// TwinCAT 3 PLC project PLC_Light_Control
// ProgramVersion: 3.1.4023.0
// libraries:
//   Tc2_BABasic, * (Beckhoff Automation GmbH)
//   Tc2_BACnetRev12, * (Beckhoff Automation GmbH)
//   Tc2_DALI, * (Beckhoff Automation GmbH)
//   Tc2_EIB, * (Beckhoff Automation GmbH)
//   Tc2_Standard, * (Beckhoff Automation GmbH)
//   Tc2_System, * (Beckhoff Automation GmbH)
//   Tc2_Utilities, * (Beckhoff Automation GmbH)
//   Tc3_Module, * (Beckhoff Automation GmbH)
// project tree:
//   / CommunicationTask.TcTTO, DimmerTask.TcTTO, PlcTask.TcTTO
//   DUTs/ E_KL6821Module.TcDUT, ST_DALI_Lamp.TcDUT
//   GVLs/ GVL_BACnet.TcGVL, GVL_GenSysInfo.TcGVL, GVL_IO.TcGVL, GVL_StreetLamps.TcGVL
//   POUs/BACnetControl/ P_BACnet_ActualLevel.TcPOU, P_BACnet_Error.TcPOU, P_BACnet_Level.TcPOU, P_BACnet_Manual.TcPOU, P_BACnet_Motion.TcPOU, P_BACnet_Scene.TcPOU
//   POUs/DimmersStreetLamps/ P_Dimmers_RB1.TcPOU, P_Dimmers_Broadcast.TcPOU, P_Dimmers_RB2.TcPOU, P_Dimmers_RB3.TcPOU
//   POUs/ FB_PBL.TcPOU, FB_SceneController.TcPOU, F_IsNight.TcPOU, MAIN.TcPOU, P_AddrAssignment.TcPOU, P_AlarmMode.TcPOU, P_AutoMode.TcPOU, P_AutoMode_Old_Broadcast.TcPOU
//   POUs/KL6821Communication/ P_DALI_RB1_Communication.TcPOU, P_DALI_RB2_Communication.TcPOU, P_DALI_RB3_Communication.TcPOU
//   POUs/KNX/ P_KNX_Communication.TcPOU, P_KNX_Data_GatesANDAlarm.TcPOU, P_KNX_Data_MotionSensors.TcPOU, P_MotionSensors.TcPOU
// real-time tasks:
//   TASK PlcTask: cycle T#10ms, priority 20, ADS port 350
//   TASK CommunicationTask: cycle T#2ms, priority 7, ADS port 351
//   TASK DimmerTask: cycle T#10ms, priority 15, ADS port 352
//   TASK Device 1 (BACnet IP)_Task_58: cycle T#40ms, priority 58, ADS port 353
//   TASK Device 1 (BACnet IP)_QueueTask: cycle T#2ms, priority 8, ADS port 354
// I/O:
//   DEVICE Device 1 (BACnet IP), AmsNetId 26.242.21.199.2.1
// variable links:
//   PLC_Light_Control Instance <-> Device 1 (BACnet IP)
//     CommunicationTask Inputs/Tc2_BACnetRev12.BACnet_Globals.fbBACnet_Adapter._AmsNetId <-> Inputs/AmsNetId
//     CommunicationTask Inputs/Tc2_BACnetRev12.BACnet_Globals.fbBACnet_Adapter._DeviceStatus <-> Inputs/Device Status
//   PLC_Light_Control Instance <-> Device 1 (BACnet IP)/Beckhoff_496669 (BACnet Server)
//     CommunicationTask Inputs/GVL_BACnet.Device._ServerStatus <-> Inputs/Server Status
//     CommunicationTask Outputs/GVL_BACnet.Device._ServerControl <-> Outputs/Server Control
//   PLC_Light_Control Instance <-> Device 1 (BACnet IP)/Beckhoff_496669 (BACnet Server)/Beckhoff_496669 (BACnet Device Object)
//     CommunicationTask Inputs/GVL_BACnet.Device._LocalDate <-> Inputs/LocalDate
//     CommunicationTask Inputs/GVL_BACnet.Device._LocalTime <-> Inputs/LocalTime
//     CommunicationTask Inputs/GVL_BACnet.Device._ObjectId <-> Inputs/ObjectIdentifier
//     CommunicationTask Inputs/GVL_BACnet.Device._SystemStatus <-> Inputs/SystemStatus
//   PLC_Light_Control Instance <-> Device 1 (BACnet IP)/Beckhoff_496669 (BACnet Server)/GVL_BACnet (BACnet Structured View Object)/fbBACnet_AV_Gates (BACnet Analog Value Object)
//     CommunicationTask Inputs/GVL_BACnet.fbBACnet_AV_Gates._PresentValue <-> Inputs/PresentValue
//     CommunicationTask Inputs/GVL_BACnet.fbBACnet_AV_Gates._StatusFlags <-> Inputs/StatusFlags
//     CommunicationTask Outputs/GVL_BACnet.fbBACnet_AV_Gates._PresentValue_Priority12 <-> Outputs/PresentValue_Priority12
//   PLC_Light_Control Instance <-> Device 1 (BACnet IP)/Beckhoff_496669 (BACnet Server)/GVL_BACnet (BACnet Structured View Object)/fbBACnet_AV_SL_ActualLevel_1 (BACnet Analog Value Object)
//     PlcTask Inputs/GVL_BACnet.fbBACnet_AV_SL_ActualLevel_1._PresentValue <-> Inputs/PresentValue
//     PlcTask Inputs/GVL_BACnet.fbBACnet_AV_SL_ActualLevel_1._StatusFlags <-> Inputs/StatusFlags
//     PlcTask Outputs/GVL_BACnet.fbBACnet_AV_SL_ActualLevel_1._PresentValue_Priority12 <-> Outputs/PresentValue_Priority12
//   PLC_Light_Control Instance <-> Device 1 (BACnet IP)/Beckhoff_496669 (BACnet Server)/GVL_BACnet (BACnet Structured View Object)/fbBACnet_AV_SL_ActualLevel_10 (BACnet Analog Value Object)
//     PlcTask Inputs/GVL_BACnet.fbBACnet_AV_SL_ActualLevel_10._PresentValue <-> Inputs/PresentValue
//     PlcTask Inputs/GVL_BACnet.fbBACnet_AV_SL_ActualLevel_10._StatusFlags <-> Inputs/StatusFlags
//     PlcTask Outputs/GVL_BACnet.fbBACnet_AV_SL_ActualLevel_10._PresentValue_Priority12 <-> Outputs/PresentValue_Priority12
//   PLC_Light_Control Instance <-> Device 1 (BACnet IP)/Beckhoff_496669 (BACnet Server)/GVL_BACnet (BACnet Structured View Object)/fbBACnet_AV_SL_ActualLevel_2 (BACnet Analog Value Object)
//     PlcTask Inputs/GVL_BACnet.fbBACnet_AV_SL_ActualLevel_2._PresentValue <-> Inputs/PresentValue
//     PlcTask Inputs/GVL_BACnet.fbBACnet_AV_SL_ActualLevel_2._StatusFlags <-> Inputs/StatusFlags
//     PlcTask Outputs/GVL_BACnet.fbBACnet_AV_SL_ActualLevel_2._PresentValue_Priority12 <-> Outputs/PresentValue_Priority12
//   PLC_Light_Control Instance <-> Device 1 (BACnet IP)/Beckhoff_496669 (BACnet Server)/GVL_BACnet (BACnet Structured View Object)/fbBACnet_AV_SL_ActualLevel_3 (BACnet Analog Value Object)
//     PlcTask Inputs/GVL_BACnet.fbBACnet_AV_SL_ActualLevel_3._PresentValue <-> Inputs/PresentValue
//     PlcTask Inputs/GVL_BACnet.fbBACnet_AV_SL_ActualLevel_3._StatusFlags <-> Inputs/StatusFlags
//     PlcTask Outputs/GVL_BACnet.fbBACnet_AV_SL_ActualLevel_3._PresentValue_Priority12 <-> Outputs/PresentValue_Priority12
//   PLC_Light_Control Instance <-> Device 1 (BACnet IP)/Beckhoff_496669 (BACnet Server)/GVL_BACnet (BACnet Structured View Object)/fbBACnet_AV_SL_ActualLevel_4 (BACnet Analog Value Object)
//     PlcTask Inputs/GVL_BACnet.fbBACnet_AV_SL_ActualLevel_4._PresentValue <-> Inputs/PresentValue
//     PlcTask Inputs/GVL_BACnet.fbBACnet_AV_SL_ActualLevel_4._StatusFlags <-> Inputs/StatusFlags
//     PlcTask Outputs/GVL_BACnet.fbBACnet_AV_SL_ActualLevel_4._PresentValue_Priority12 <-> Outputs/PresentValue_Priority12
//   PLC_Light_Control Instance <-> Device 1 (BACnet IP)/Beckhoff_496669 (BACnet Server)/GVL_BACnet (BACnet Structured View Object)/fbBACnet_AV_SL_ActualLevel_5 (BACnet Analog Value Object)
//     PlcTask Inputs/GVL_BACnet.fbBACnet_AV_SL_ActualLevel_5._PresentValue <-> Inputs/PresentValue
//     PlcTask Inputs/GVL_BACnet.fbBACnet_AV_SL_ActualLevel_5._StatusFlags <-> Inputs/StatusFlags
//     PlcTask Outputs/GVL_BACnet.fbBACnet_AV_SL_ActualLevel_5._PresentValue_Priority12 <-> Outputs/PresentValue_Priority12
//   PLC_Light_Control Instance <-> Device 1 (BACnet IP)/Beckhoff_496669 (BACnet Server)/GVL_BACnet (BACnet Structured View Object)/fbBACnet_AV_SL_ActualLevel_6 (BACnet Analog Value Object)
//     PlcTask Inputs/GVL_BACnet.fbBACnet_AV_SL_ActualLevel_6._PresentValue <-> Inputs/PresentValue
//     PlcTask Inputs/GVL_BACnet.fbBACnet_AV_SL_ActualLevel_6._StatusFlags <-> Inputs/StatusFlags
//     PlcTask Outputs/GVL_BACnet.fbBACnet_AV_SL_ActualLevel_6._PresentValue_Priority12 <-> Outputs/PresentValue_Priority12
//   PLC_Light_Control Instance <-> Device 1 (BACnet IP)/Beckhoff_496669 (BACnet Server)/GVL_BACnet (BACnet Structured View Object)/fbBACnet_AV_SL_ActualLevel_7 (BACnet Analog Value Object)
//     PlcTask Inputs/GVL_BACnet.fbBACnet_AV_SL_ActualLevel_7._PresentValue <-> Inputs/PresentValue
//     PlcTask Inputs/GVL_BACnet.fbBACnet_AV_SL_ActualLevel_7._StatusFlags <-> Inputs/StatusFlags
//     PlcTask Outputs/GVL_BACnet.fbBACnet_AV_SL_ActualLevel_7._PresentValue_Priority12 <-> Outputs/PresentValue_Priority12
//   PLC_Light_Control Instance <-> Device 1 (BACnet IP)/Beckhoff_496669 (BACnet Server)/GVL_BACnet (BACnet Structured View Object)/fbBACnet_AV_SL_ActualLevel_8 (BACnet Analog Value Object)
//     PlcTask Inputs/GVL_BACnet.fbBACnet_AV_SL_ActualLevel_8._PresentValue <-> Inputs/PresentValue
//     PlcTask Inputs/GVL_BACnet.fbBACnet_AV_SL_ActualLevel_8._StatusFlags <-> Inputs/StatusFlags
//     PlcTask Outputs/GVL_BACnet.fbBACnet_AV_SL_ActualLevel_8._PresentValue_Priority12 <-> Outputs/PresentValue_Priority12
//   PLC_Light_Control Instance <-> Device 1 (BACnet IP)/Beckhoff_496669 (BACnet Server)/GVL_BACnet (BACnet Structured View Object)/fbBACnet_AV_SL_ActualLevel_9 (BACnet Analog Value Object)
//     PlcTask Inputs/GVL_BACnet.fbBACnet_AV_SL_ActualLevel_9._PresentValue <-> Inputs/PresentValue
//     PlcTask Inputs/GVL_BACnet.fbBACnet_AV_SL_ActualLevel_9._StatusFlags <-> Inputs/StatusFlags
//     PlcTask Outputs/GVL_BACnet.fbBACnet_AV_SL_ActualLevel_9._PresentValue_Priority12 <-> Outputs/PresentValue_Priority12
//   PLC_Light_Control Instance <-> Device 1 (BACnet IP)/Beckhoff_496669 (BACnet Server)/GVL_BACnet (BACnet Structured View Object)/fbBACnet_AV_SL_Error (BACnet Analog Value Object)
//     PlcTask Inputs/GVL_BACnet.fbBACnet_AV_SL_Error._PresentValue <-> Inputs/PresentValue
//     PlcTask Inputs/GVL_BACnet.fbBACnet_AV_SL_Error._StatusFlags <-> Inputs/StatusFlags
//     PlcTask Outputs/GVL_BACnet.fbBACnet_AV_SL_Error._PresentValue_Priority12 <-> Outputs/PresentValue_Priority12
//   PLC_Light_Control Instance <-> Device 1 (BACnet IP)/Beckhoff_496669 (BACnet Server)/GVL_BACnet (BACnet Structured View Object)/fbBACnet_AV_SL_Level_1 (BACnet Analog Value Object)
//     PlcTask Inputs/GVL_BACnet.fbBACnet_AV_SL_Level_1._PresentValue <-> Inputs/PresentValue
//     PlcTask Inputs/GVL_BACnet.fbBACnet_AV_SL_Level_1._StatusFlags <-> Inputs/StatusFlags
//     PlcTask Outputs/GVL_BACnet.fbBACnet_AV_SL_Level_1._PresentValue_Priority12 <-> Outputs/PresentValue_Priority12
//   PLC_Light_Control Instance <-> Device 1 (BACnet IP)/Beckhoff_496669 (BACnet Server)/GVL_BACnet (BACnet Structured View Object)/fbBACnet_AV_SL_Level_10 (BACnet Analog Value Object)
//     PlcTask Inputs/GVL_BACnet.fbBACnet_AV_SL_Level_10._PresentValue <-> Inputs/PresentValue
//     PlcTask Inputs/GVL_BACnet.fbBACnet_AV_SL_Level_10._StatusFlags <-> Inputs/StatusFlags
//     PlcTask Outputs/GVL_BACnet.fbBACnet_AV_SL_Level_10._PresentValue_Priority12 <-> Outputs/PresentValue_Priority12
//   PLC_Light_Control Instance <-> Device 1 (BACnet IP)/Beckhoff_496669 (BACnet Server)/GVL_BACnet (BACnet Structured View Object)/fbBACnet_AV_SL_Level_2 (BACnet Analog Value Object)
//     PlcTask Inputs/GVL_BACnet.fbBACnet_AV_SL_Level_2._PresentValue <-> Inputs/PresentValue
//     PlcTask Inputs/GVL_BACnet.fbBACnet_AV_SL_Level_2._StatusFlags <-> Inputs/StatusFlags
//     PlcTask Outputs/GVL_BACnet.fbBACnet_AV_SL_Level_2._PresentValue_Priority12 <-> Outputs/PresentValue_Priority12
//   PLC_Light_Control Instance <-> Device 1 (BACnet IP)/Beckhoff_496669 (BACnet Server)/GVL_BACnet (BACnet Structured View Object)/fbBACnet_AV_SL_Level_3 (BACnet Analog Value Object)
//     PlcTask Inputs/GVL_BACnet.fbBACnet_AV_SL_Level_3._PresentValue <-> Inputs/PresentValue
//     PlcTask Inputs/GVL_BACnet.fbBACnet_AV_SL_Level_3._StatusFlags <-> Inputs/StatusFlags
//     PlcTask Outputs/GVL_BACnet.fbBACnet_AV_SL_Level_3._PresentValue_Priority12 <-> Outputs/PresentValue_Priority12
//   PLC_Light_Control Instance <-> Device 1 (BACnet IP)/Beckhoff_496669 (BACnet Server)/GVL_BACnet (BACnet Structured View Object)/fbBACnet_AV_SL_Level_4 (BACnet Analog Value Object)
//     PlcTask Inputs/GVL_BACnet.fbBACnet_AV_SL_Level_4._PresentValue <-> Inputs/PresentValue
//     PlcTask Inputs/GVL_BACnet.fbBACnet_AV_SL_Level_4._StatusFlags <-> Inputs/StatusFlags
//     PlcTask Outputs/GVL_BACnet.fbBACnet_AV_SL_Level_4._PresentValue_Priority12 <-> Outputs/PresentValue_Priority12
//   PLC_Light_Control Instance <-> Device 1 (BACnet IP)/Beckhoff_496669 (BACnet Server)/GVL_BACnet (BACnet Structured View Object)/fbBACnet_AV_SL_Level_5 (BACnet Analog Value Object)
//     PlcTask Inputs/GVL_BACnet.fbBACnet_AV_SL_Level_5._PresentValue <-> Inputs/PresentValue
//     PlcTask Inputs/GVL_BACnet.fbBACnet_AV_SL_Level_5._StatusFlags <-> Inputs/StatusFlags
//     PlcTask Outputs/GVL_BACnet.fbBACnet_AV_SL_Level_5._PresentValue_Priority12 <-> Outputs/PresentValue_Priority12
//   PLC_Light_Control Instance <-> Device 1 (BACnet IP)/Beckhoff_496669 (BACnet Server)/GVL_BACnet (BACnet Structured View Object)/fbBACnet_AV_SL_Level_6 (BACnet Analog Value Object)
//     PlcTask Inputs/GVL_BACnet.fbBACnet_AV_SL_Level_6._PresentValue <-> Inputs/PresentValue
//     PlcTask Inputs/GVL_BACnet.fbBACnet_AV_SL_Level_6._StatusFlags <-> Inputs/StatusFlags
//     PlcTask Outputs/GVL_BACnet.fbBACnet_AV_SL_Level_6._PresentValue_Priority12 <-> Outputs/PresentValue_Priority12
//   PLC_Light_Control Instance <-> Device 1 (BACnet IP)/Beckhoff_496669 (BACnet Server)/GVL_BACnet (BACnet Structured View Object)/fbBACnet_AV_SL_Level_7 (BACnet Analog Value Object)
//     PlcTask Inputs/GVL_BACnet.fbBACnet_AV_SL_Level_7._PresentValue <-> Inputs/PresentValue
//     PlcTask Inputs/GVL_BACnet.fbBACnet_AV_SL_Level_7._StatusFlags <-> Inputs/StatusFlags
//     PlcTask Outputs/GVL_BACnet.fbBACnet_AV_SL_Level_7._PresentValue_Priority12 <-> Outputs/PresentValue_Priority12
//   PLC_Light_Control Instance <-> Device 1 (BACnet IP)/Beckhoff_496669 (BACnet Server)/GVL_BACnet (BACnet Structured View Object)/fbBACnet_AV_SL_Level_8 (BACnet Analog Value Object)
//     PlcTask Inputs/GVL_BACnet.fbBACnet_AV_SL_Level_8._PresentValue <-> Inputs/PresentValue
//     PlcTask Inputs/GVL_BACnet.fbBACnet_AV_SL_Level_8._StatusFlags <-> Inputs/StatusFlags
//     PlcTask Outputs/GVL_BACnet.fbBACnet_AV_SL_Level_8._PresentValue_Priority12 <-> Outputs/PresentValue_Priority12
//   PLC_Light_Control Instance <-> Device 1 (BACnet IP)/Beckhoff_496669 (BACnet Server)/GVL_BACnet (BACnet Structured View Object)/fbBACnet_AV_SL_Level_9 (BACnet Analog Value Object)
//     PlcTask Inputs/GVL_BACnet.fbBACnet_AV_SL_Level_9._PresentValue <-> Inputs/PresentValue
//     PlcTask Inputs/GVL_BACnet.fbBACnet_AV_SL_Level_9._StatusFlags <-> Inputs/StatusFlags
//     PlcTask Outputs/GVL_BACnet.fbBACnet_AV_SL_Level_9._PresentValue_Priority12 <-> Outputs/PresentValue_Priority12
//   PLC_Light_Control Instance <-> Device 1 (BACnet IP)/Beckhoff_496669 (BACnet Server)/GVL_BACnet (BACnet Structured View Object)/fbBACnet_AV_SL_Manual (BACnet Analog Value Object)
//     PlcTask Inputs/GVL_BACnet.fbBACnet_AV_SL_Manual._PresentValue <-> Inputs/PresentValue
//     PlcTask Inputs/GVL_BACnet.fbBACnet_AV_SL_Manual._StatusFlags <-> Inputs/StatusFlags
//     PlcTask Outputs/GVL_BACnet.fbBACnet_AV_SL_Manual._PresentValue_Priority12 <-> Outputs/PresentValue_Priority12
//   PLC_Light_Control Instance <-> Device 1 (BACnet IP)/Beckhoff_496669 (BACnet Server)/GVL_BACnet (BACnet Structured View Object)/fbBACnet_AV_SL_Motion (BACnet Analog Value Object)
//     PlcTask Inputs/GVL_BACnet.fbBACnet_AV_SL_Motion._PresentValue <-> Inputs/PresentValue
//     PlcTask Inputs/GVL_BACnet.fbBACnet_AV_SL_Motion._StatusFlags <-> Inputs/StatusFlags
//     PlcTask Outputs/GVL_BACnet.fbBACnet_AV_SL_Motion._PresentValue_Priority12 <-> Outputs/PresentValue_Priority12
//   PLC_Light_Control Instance <-> Device 1 (BACnet IP)/Beckhoff_496669 (BACnet Server)/GVL_BACnet (BACnet Structured View Object)/fbBACnet_AV_SL_Scene (BACnet Analog Value Object)
//     PlcTask Inputs/GVL_BACnet.fbBACnet_AV_SL_Scene._PresentValue <-> Inputs/PresentValue
//     PlcTask Inputs/GVL_BACnet.fbBACnet_AV_SL_Scene._StatusFlags <-> Inputs/StatusFlags
//     PlcTask Outputs/GVL_BACnet.fbBACnet_AV_SL_Scene._PresentValue_Priority12 <-> Outputs/PresentValue_Priority12
//   PLC_Light_Control Instance <-> Device 1 (BACnet IP)/Beckhoff_496669 (BACnet Server)/GVL_BACnet (BACnet Structured View Object)/fbBACnet_BV_Alarm (BACnet Binary Value Object)
//     CommunicationTask Inputs/GVL_BACnet.fbBACnet_BV_Alarm._PresentValue <-> Inputs/PresentValue
//     CommunicationTask Inputs/GVL_BACnet.fbBACnet_BV_Alarm._StatusFlags <-> Inputs/StatusFlags
//     CommunicationTask Outputs/GVL_BACnet.fbBACnet_BV_Alarm._PresentValue_Priority12 <-> Outputs/PresentValue_Priority12

CONFIGURATION PLC_Light_Control
    RESOURCE PLC ON TwinCAT3
        TASK CommunicationTask(INTERVAL := T#2ms, PRIORITY := 7);
        TASK DimmerTask(INTERVAL := T#10ms, PRIORITY := 15);
        TASK PlcTask(INTERVAL := T#10ms, PRIORITY := 20);
        PROGRAM P_DALI_RB1_Communication WITH CommunicationTask : P_DALI_RB1_Communication;
        PROGRAM P_DALI_RB2_Communication WITH CommunicationTask : P_DALI_RB2_Communication;
        PROGRAM P_DALI_RB3_Communication WITH CommunicationTask : P_DALI_RB3_Communication;
        PROGRAM P_KNX_Communication WITH CommunicationTask : P_KNX_Communication;
        PROGRAM P_KNX_Data_MotionSensors WITH CommunicationTask : P_KNX_Data_MotionSensors;
        PROGRAM P_KNX_Data_GatesANDAlarm WITH CommunicationTask : P_KNX_Data_GatesANDAlarm;
        PROGRAM P_Dimmers_RB1 WITH DimmerTask : P_Dimmers_RB1;
        PROGRAM P_Dimmers_RB2 WITH DimmerTask : P_Dimmers_RB2;
        PROGRAM P_Dimmers_RB3 WITH DimmerTask : P_Dimmers_RB3;
        PROGRAM P_Dimmers_Broadcast WITH DimmerTask : P_Dimmers_Broadcast;
        PROGRAM MAIN WITH PlcTask : MAIN;
    END_RESOURCE
END_CONFIGURATION

// ---- DUTs/E_KL6821Module.TcDUT
//{attribute 'qualified_only'}
//{attribute 'strict'}
TYPE E_KL6821Module :
(
	eKL6821Module_none	:= 0,
	eKL6821Module_RB1 	:= 10,
	eKL6821Module_RB2	:= 20,
	eKL6821Module_RB3	:= 30
	
);
END_TYPE

// ---- DUTs/ST_DALI_Lamp.TcDUT
TYPE ST_DALI_Lamp :
STRUCT
	bManualCtrl		: BOOL;		// if TRUE scenes do not apply
	bLampFailure	: BOOL;		// if TRUE ballast has a lamp problem
	
	nStatus			: BYTE;		// status of a ballast
	
	nLevel			: BYTE;		// 0-255
	
	eKL6821Module	: E_KL6821Module;	//DALI module to which Lamp is connected
	nAddrShort1		: BYTE;				//first 	DALI gear address
	nAddrShort2		: BYTE;				//second 	DALI gear address 
	
	ref_stCommandBuffer	: REFERENCE TO ST_DALIV2CommandBuffer;	//reference to command buffer
	
	//group addresses which DALI_Lamp belongs to
	arrAddrGroup	: ARRAY [1..4] OF BYTE;
	
	//sensors
	bMotionSensor	AT%I*	: BOOL;	//direct info from sensor, edge means movement occured
	bMotionFlag				: BOOL;	//flag keeping info about motion as TRUE for specified period of time
	
END_STRUCT
END_TYPE

// ---- GVLs/GVL_BACnet.TcGVL
VAR_GLOBAL
	Device				: FB_BACnet_Device;
	
	// "SL" means - "Streat Lamps"
	
	
	// binary value object
	fbBACnet_BV_Alarm			:FB_BACnet_BinaryValue;			(* ~ (BACnet_ObjectIdentifier	:  100   : NOLINK) *)
	
	//other signals than lamps
	//gates pseuda-array
	fbBACnet_AV_Gates			:FB_BACnet_AnalogValue;			(* ~ (BACnet_ObjectIdentifier	:  200   : NOLINK) *)
	
	// pseudo-arrays - multiple BVs in one BACnet AV object,
	// bit-wise informations - each bit corresponds to particular lamp 
	fbBACnet_AV_SL_Manual		: FB_BACnet_AnalogValue;		(* ~ (BACnet_ObjectIdentifier	: 1111   : NOLINK) *)
	bBACnet_ResetManual			: BOOL;
	
	fbBACnet_AV_SL_Scene		: FB_BACnet_AnalogValue;		(* ~ (BACnet_ObjectIdentifier	: 2222   : NOLINK) *)								
	fbBACnet_AV_SL_Motion		: FB_BACnet_AnalogValue;		(* ~ (BACnet_ObjectIdentifier	: 3333   : NOLINK) *)
	fbBACnet_AV_SL_Error		: FB_BACnet_AnalogValue;		(* ~ (BACnet_ObjectIdentifier	: 9999   : NOLINK) *)
	
	// one variable one BACnet object
	fbBACnet_AV_SL_Level_1		: FB_BACnet_AnalogValue;	(* ~ (BACnet_ObjectIdentifier	: 4001   : NOLINK) *)
	fbBACnet_AV_SL_Level_2		: FB_BACnet_AnalogValue;	(* ~ (BACnet_ObjectIdentifier	: 4002   : NOLINK) *)
	fbBACnet_AV_SL_Level_3		: FB_BACnet_AnalogValue;	(* ~ (BACnet_ObjectIdentifier	: 4003   : NOLINK) *)
	fbBACnet_AV_SL_Level_4		: FB_BACnet_AnalogValue;	(* ~ (BACnet_ObjectIdentifier	: 4004   : NOLINK) *)
	fbBACnet_AV_SL_Level_5		: FB_BACnet_AnalogValue;	(* ~ (BACnet_ObjectIdentifier	: 4005   : NOLINK) *)
	fbBACnet_AV_SL_Level_6		: FB_BACnet_AnalogValue;	(* ~ (BACnet_ObjectIdentifier	: 4006   : NOLINK) *)
	fbBACnet_AV_SL_Level_7		: FB_BACnet_AnalogValue;	(* ~ (BACnet_ObjectIdentifier	: 4007   : NOLINK) *)
	fbBACnet_AV_SL_Level_8		: FB_BACnet_AnalogValue;	(* ~ (BACnet_ObjectIdentifier	: 4008   : NOLINK) *)
	fbBACnet_AV_SL_Level_9		: FB_BACnet_AnalogValue;	(* ~ (BACnet_ObjectIdentifier	: 4009   : NOLINK) *)
	fbBACnet_AV_SL_Level_10		: FB_BACnet_AnalogValue;	(* ~ (BACnet_ObjectIdentifier	: 4010   : NOLINK) *)
	
	fbBACnet_AV_SL_ActualLevel_1		: FB_BACnet_AnalogValue;	(* ~ (BACnet_ObjectIdentifier	: 5001   : NOLINK) *)
	fbBACnet_AV_SL_ActualLevel_2		: FB_BACnet_AnalogValue;	(* ~ (BACnet_ObjectIdentifier	: 5002   : NOLINK) *)
	fbBACnet_AV_SL_ActualLevel_3		: FB_BACnet_AnalogValue;	(* ~ (BACnet_ObjectIdentifier	: 5003   : NOLINK) *)
	fbBACnet_AV_SL_ActualLevel_4		: FB_BACnet_AnalogValue;	(* ~ (BACnet_ObjectIdentifier	: 5004   : NOLINK) *)
	fbBACnet_AV_SL_ActualLevel_5		: FB_BACnet_AnalogValue;	(* ~ (BACnet_ObjectIdentifier	: 5005   : NOLINK) *)
	fbBACnet_AV_SL_ActualLevel_6		: FB_BACnet_AnalogValue;	(* ~ (BACnet_ObjectIdentifier	: 5006   : NOLINK) *)
	fbBACnet_AV_SL_ActualLevel_7		: FB_BACnet_AnalogValue;	(* ~ (BACnet_ObjectIdentifier	: 5007   : NOLINK) *)
	fbBACnet_AV_SL_ActualLevel_8		: FB_BACnet_AnalogValue;	(* ~ (BACnet_ObjectIdentifier	: 5008   : NOLINK) *)
	fbBACnet_AV_SL_ActualLevel_9		: FB_BACnet_AnalogValue;	(* ~ (BACnet_ObjectIdentifier	: 5009   : NOLINK) *)
	fbBACnet_AV_SL_ActualLevel_10		: FB_BACnet_AnalogValue;	(* ~ (BACnet_ObjectIdentifier	: 5010   : NOLINK) *)

END_VAR

// ---- GVLs/GVL_GenSysInfo.TcGVL
VAR_GLOBAL
	tMotionSensorsTOF_PT		: TIME := T#5M;			//how long lamps stay lighten up after move ended
	tMotionSensorsTOF_info_PT	: TIME := T#10S;		//how long motion flags stay TRUE after move ended
	todGlobalTime				: TOD := TOD#10:0:0;
END_VAR

VAR_GLOBAL CONSTANT
	
	byStreetLampsCount			: BYTE := 10;
	byStreetLampsScenesNumber	: BYTE := 40;
	
	//Standard Brightness
	
	c_byBrightness_Alarm	: BYTE := 254;
	c_byBrightness_Motion	: BYTE := 230;
	c_byBrightness_Night	: BYTE := 180;
	c_byBrightness_Day		: BYTE := 0; 
	
	
	
END_VAR

// ---- GVLs/GVL_IO.TcGVL
{attribute 'qualified_only'}
VAR_GLOBAL
	
	//DALI Communication variables
	
		//RB1
		stKL6821InData_RB1		AT%I*	: ST_KL6821InData;
		stKL6821OutData_RB1		AT%Q*	: ST_KL6821OutData;
		stCommandBuffer_RB1				: ST_DALIV2CommandBuffer;
		//RB2
		stKL6821InData_RB2		AT%I*	: ST_KL6821InData;
		stKL6821OutData_RB2		AT%Q*	: ST_KL6821OutData;
		stCommandBuffer_RB2				: ST_DALIV2CommandBuffer;
		//RB3
		stKL6821InData_RB3		AT%I*	: ST_KL6821InData;
		stKL6821OutData_RB3		AT%Q*	: ST_KL6821OutData;
		stCommandBuffer_RB3				: ST_DALIV2CommandBuffer;
	
	//KNX Communication
		
		//KL6301
		KL6301_IN             	AT%I*	: ARRAY [1..24] OF BYTE;
		KL6301_OUT            	AT%Q*	: ARRAY [1..24] OF BYTE;
		str_Data_Rec          			: EIB_REC;
		
	//Other
		
		//street lamp that has no DALI
		//therefore it is controlled via digital output (DO)
		bStreetLamp_DO1			AT%Q*	: BOOL;
		
END_VAR

VAR_GLOBAL PERSISTENT
	
	//DALI Gears
		
		//Street Lamps
		arrStreetLamps			: ARRAY [1..byStreetLampsCount] OF ST_DALI_Lamp;
	
	//DALI Scenes
		
		//Street Lamps
		arrScenesStreetLampsLevels	: ARRAY [1..byStreetLampsScenesNumber, 1..byStreetLampsCount] OF BYTE;	//specifies lamp level in a scene
		
		
END_VAR

// ---- GVLs/GVL_StreetLamps.TcGVL
{attribute 'qualified_only'}
VAR_GLOBAL
	
	//Addres Short
	bSetDimmValue					: BOOL := FALSE;
	                            	
	tSwitchOverTime					: TIME := T#400MS;
	bMemoryModeOn					: BOOL := FALSE;
	nOnValueWithoutMemoryMode		: BYTE := 254;
	nMasterDevAddr              	: BYTE := 0;
	tCycleActualLevelMasterDev  	: TIME := T#0S;
	
	//Addres Broadcast
	bSetDimmValue_B					: BOOL := FALSE;
	nDimmValue_B					: BYTE;
	                            	
	tSwitchOverTime_B				: TIME := T#400MS;
	bMemoryModeOn_B					: BOOL := FALSE;
	nOnValueWithoutMemoryMode_B		: BYTE := 254;
	nMasterDevAddr_B              	: BYTE := 0;
	tCycleActualLevelMasterDev_B 	: TIME := T#0S;
END_VAR

// ---- POUs/KL6821Communication/P_DALI_RB1_Communication.TcPOU
PROGRAM P_DALI_RB1_Communication
VAR
	//INPUTS
	fbKL6821Communication		: FB_KL6821Communication;
	bResetMaximumDemandCounter	: BOOL;
	bResetOverflowCounter		: BOOL;
	bResetInactiveProcessImage	: BOOL;
	nOptions					: DWORD;
	
	//VAR_IN_OUT
	//--- See GVL_IO ---
	
	//OUTPUTS
	bBusy						: BOOL;
	bError						: BOOL;
	nErrorId					: UDINT;
	arrBufferDemandMeter		: ARRAY [0..2] OF BYTE;
	arrBufferMaximumDemandMeter	: ARRAY [0..2] OF BYTE;
	arrBufferOverflowCounter	: ARRAY [0..2] OF UINT;
	bLineIsBusy					: BOOL;
	bLineIsInitialized			: BOOL;
	bDigitalInput1Active		: BOOL;
	bDigitalInput2Active		: BOOL;
	bProcessImageInactive		: BOOL;
	bCollisionError				: BOOL;
	bPowerSupplyError			: BOOL;
	bShortCircuit				: BOOL;
END_VAR

fbKL6821Communication(
    bResetMaximumDemandCounter := bResetMaximumDemandCounter,
    bResetOverflowCounter := bResetOverflowCounter,
    bResetInactiveProcessImage := bResetInactiveProcessImage,
    nOptions := nOptions,
    stInData := GVL_IO.stKL6821InData_RB1,
    stOutData := GVL_IO.stKL6821OutData_RB1,
    stCommandBuffer := GVL_IO.stCommandBuffer_RB1); // FB_KL6821Communication
bBusy := fbKL6821Communication.bBusy;
bError := fbKL6821Communication.bError;
nErrorId := fbKL6821Communication.nErrorId;
arrBufferDemandMeter := fbKL6821Communication.arrBufferDemandMeter;
arrBufferMaximumDemandMeter := fbKL6821Communication.arrBufferMaximumDemandMeter;
arrBufferOverflowCounter := fbKL6821Communication.arrBufferOverflowCounter;
bLineIsBusy := fbKL6821Communication.bLineIsBusy;
bLineIsInitialized := fbKL6821Communication.bLineIsInitialized;
bDigitalInput1Active := fbKL6821Communication.bDigitalInput1Active;
bDigitalInput2Active := fbKL6821Communication.bDigitalInput2Active;
bProcessImageInactive := fbKL6821Communication.bProcessImageInactive;
bCollisionError := fbKL6821Communication.bCollisionError;
bPowerSupplyError := fbKL6821Communication.bPowerSupplyError;
bShortCircuit := fbKL6821Communication.bShortCircuit;

END_PROGRAM

// ---- POUs/KL6821Communication/P_DALI_RB2_Communication.TcPOU
PROGRAM P_DALI_RB2_Communication
VAR
	//INPUTS
	fbKL6821Communication		: FB_KL6821Communication;
	bResetMaximumDemandCounter	: BOOL;
	bResetOverflowCounter		: BOOL;
	bResetInactiveProcessImage	: BOOL;
	nOptions					: DWORD;
	
	//VAR_IN_OUT
	//--- See GVL_IO ---
	
	//OUTPUTS
	bBusy						: BOOL;
	bError						: BOOL;
	nErrorId					: UDINT;
	arrBufferDemandMeter		: ARRAY [0..2] OF BYTE;
	arrBufferMaximumDemandMeter	: ARRAY [0..2] OF BYTE;
	arrBufferOverflowCounter	: ARRAY [0..2] OF UINT;
	bLineIsBusy					: BOOL;
	bLineIsInitialized			: BOOL;
	bDigitalInput1Active		: BOOL;
	bDigitalInput2Active		: BOOL;
	bProcessImageInactive		: BOOL;
	bCollisionError				: BOOL;
	bPowerSupplyError			: BOOL;
	bShortCircuit				: BOOL;
END_VAR

fbKL6821Communication(
    bResetMaximumDemandCounter := bResetMaximumDemandCounter,
    bResetOverflowCounter := bResetOverflowCounter,
    bResetInactiveProcessImage := bResetInactiveProcessImage,
    nOptions := nOptions,
    stInData := GVL_IO.stKL6821InData_RB2,
    stOutData := GVL_IO.stKL6821OutData_RB2,
    stCommandBuffer := GVL_IO.stCommandBuffer_RB2); // FB_KL6821Communication
bBusy := fbKL6821Communication.bBusy;
bError := fbKL6821Communication.bError;
nErrorId := fbKL6821Communication.nErrorId;
arrBufferDemandMeter := fbKL6821Communication.arrBufferDemandMeter;
arrBufferMaximumDemandMeter := fbKL6821Communication.arrBufferMaximumDemandMeter;
arrBufferOverflowCounter := fbKL6821Communication.arrBufferOverflowCounter;
bLineIsBusy := fbKL6821Communication.bLineIsBusy;
bLineIsInitialized := fbKL6821Communication.bLineIsInitialized;
bDigitalInput1Active := fbKL6821Communication.bDigitalInput1Active;
bDigitalInput2Active := fbKL6821Communication.bDigitalInput2Active;
bProcessImageInactive := fbKL6821Communication.bProcessImageInactive;
bCollisionError := fbKL6821Communication.bCollisionError;
bPowerSupplyError := fbKL6821Communication.bPowerSupplyError;
bShortCircuit := fbKL6821Communication.bShortCircuit;

END_PROGRAM

// ---- POUs/KL6821Communication/P_DALI_RB3_Communication.TcPOU
PROGRAM P_DALI_RB3_Communication
VAR
	//INPUTS
	fbKL6821Communication		: FB_KL6821Communication;
	bResetMaximumDemandCounter	: BOOL;
	bResetOverflowCounter		: BOOL;
	bResetInactiveProcessImage	: BOOL;
	nOptions					: DWORD;
	
	//VAR_IN_OUT
	//--- See GVL_IO ---
	
	//OUTPUTS
	bBusy						: BOOL;
	bError						: BOOL;
	nErrorId					: UDINT;
	arrBufferDemandMeter		: ARRAY [0..2] OF BYTE;
	arrBufferMaximumDemandMeter	: ARRAY [0..2] OF BYTE;
	arrBufferOverflowCounter	: ARRAY [0..2] OF UINT;
	bLineIsBusy					: BOOL;
	bLineIsInitialized			: BOOL;
	bDigitalInput1Active		: BOOL;
	bDigitalInput2Active		: BOOL;
	bProcessImageInactive		: BOOL;
	bCollisionError				: BOOL;
	bPowerSupplyError			: BOOL;
	bShortCircuit				: BOOL;
END_VAR

fbKL6821Communication(
    bResetMaximumDemandCounter := bResetMaximumDemandCounter,
    bResetOverflowCounter := bResetOverflowCounter,
    bResetInactiveProcessImage := bResetInactiveProcessImage,
    nOptions := nOptions,
    stInData := GVL_IO.stKL6821InData_RB3,
    stOutData := GVL_IO.stKL6821OutData_RB3,
    stCommandBuffer := GVL_IO.stCommandBuffer_RB3); // FB_KL6821Communication
bBusy := fbKL6821Communication.bBusy;
bError := fbKL6821Communication.bError;
nErrorId := fbKL6821Communication.nErrorId;
arrBufferDemandMeter := fbKL6821Communication.arrBufferDemandMeter;
arrBufferMaximumDemandMeter := fbKL6821Communication.arrBufferMaximumDemandMeter;
arrBufferOverflowCounter := fbKL6821Communication.arrBufferOverflowCounter;
bLineIsBusy := fbKL6821Communication.bLineIsBusy;
bLineIsInitialized := fbKL6821Communication.bLineIsInitialized;
bDigitalInput1Active := fbKL6821Communication.bDigitalInput1Active;
bDigitalInput2Active := fbKL6821Communication.bDigitalInput2Active;
bProcessImageInactive := fbKL6821Communication.bProcessImageInactive;
bCollisionError := fbKL6821Communication.bCollisionError;
bPowerSupplyError := fbKL6821Communication.bPowerSupplyError;
bShortCircuit := fbKL6821Communication.bShortCircuit;

END_PROGRAM

// ---- POUs/KNX/P_KNX_Communication.TcPOU
PROGRAM P_KNX_Communication
VAR
	KL6301_0: KL6301;
	
	bActivate             : BOOL := TRUE;
	idx                   : INT := 1;
	EIB_PHYS_ADDR         : EIB_PHYS_ADDR := (Area := 1, Line := 6, Device := 150);
	EIB_GROUP_FILTER      : ARRAY [1..8] OF EIB_GROUP_FILTER := [
																	(GROUP_ADDR := (MAIN := 12, SUB_MAIN := 0, NUMBER := 0),
																	 GROUP_LEN  := 63),
																	(GROUP_ADDR := (MAIN := 12, SUB_MAIN := 1, NUMBER := 0),
																	 GROUP_LEN  := 63)
																];
	iMode                 : INT := 0;
	tTimeout              : TIME := T#5S;
	
	bActive               : BOOL;
	bReady                : BOOL;
	bError                : BOOL;
	iErrorId              : EIB_Error_Code;
	
END_VAR

KL6301_0(
    bActivate := bActivate,
    idx := idx,
    EIB_PHYS_ADDR := EIB_PHYS_ADDR,
    EIB_GROUP_FILTER := EIB_GROUP_FILTER,
    iMode := iMode,
    tTimeout := tTimeout,
    KL6301_IN := GVL_IO.KL6301_IN,
    KL6301_OUT := GVL_IO.KL6301_OUT); // KL6301
bActive := KL6301_0.bActive;
bReady := KL6301_0.bReady;
bError := KL6301_0.bError;
iErrorId := KL6301_0.iErrorId;
GVL_IO.str_Data_Rec := KL6301_0.str_Data_Rec;

END_PROGRAM

// ---- POUs/MAIN.TcPOU
PROGRAM MAIN
VAR
	tonCycle			: TON; //timer used to measure 1min period
	fbSceneController	: FB_SceneController;
	fbPBL				: FB_PBL; //previous brightness level data block
END_VAR

//init timer and set dimm value for all street lamps every 1M
//in other words: repeat control signal in case of power failure
tonCycle(IN := NOT tonCycle.Q, PT:=T#1M, Q=>GVL_StreetLamps.bSetDimmValue);

//assign DALI addresses at the begining of the program
P_AddrAssignment();

//P_BACnet_ActualLevel();
//P_BACnet_Error();
//P_BACnet_Level();
//P_BACnet_Manual();
//P_BACnet_Motion();
//P_BACnet_Scene();

//KNX motion sensors activated
P_MotionSensors(bEnable := TRUE);

//listen to alarm
P_AlarmMode();

//if there is no alarm
IF NOT fbBACnet_BV_Alarm.bPresentValue THEN
	//maintain auto mode and scene control
	P_AutoMode();
	fbSceneController();
END_IF

END_PROGRAM

// ---- POUs/FB_SceneController.TcPOU
(*
Funion block manages the scene data. When rising edge on bSceneON is detected
it recalls a scene from the memory. If rising edge is detected on bSaveScene
it saves the scene to memory under bySceneID number.
Futhermore it save the information about individual lamps being cut off from the scene.
Main idea is that FB uses GVL_IO.arrStreetLamps as 'live buffer' ,
GVL_IO.arrScenes<  > on the other hand is a data 'memory buffer'. 
*)
FUNCTION_BLOCK FB_SceneController
VAR_INPUT
END_VAR
VAR_OUTPUT
	bBusy				:BOOL:=FALSE;		//when TRUE FB is busy working
END_VAR
VAR
	bySceneID			: BYTE;		//number of scene that is being manipulated
	iSelector			: INT := 0;	//variable used in CASE statement
	iCounter			: INT := 0;	//for loop counter
	
	
END_VAR

//if FB is not busy
IF NOT bBusy THEN
	//read BACnet object
	iSelector := REAL_TO_INT(fbBACnet_AV_SL_Scene.fPresentValue);
END_IF

CASE iSelector OF
	0, 255:	//idle state
		;
		
	1..127:	//SceneON
		bBusy := TRUE;	//set a flag indicating that this FB is busy
		
		//reset manual mode
		bBACnet_ResetManual := TRUE;
		
		//convert int to byte
		bySceneID := INT_TO_BYTE(iSelector);
		
		//rewrite power levels from memory buffer to BACnet objects
		fbBACnet_AV_SL_Level_1.fPV  := GVL_IO.arrScenesStreetLampsLevels[bySceneID, 1];
		fbBACnet_AV_SL_Level_2.fPV  := GVL_IO.arrScenesStreetLampsLevels[bySceneID, 2];
		fbBACnet_AV_SL_Level_3.fPV  := GVL_IO.arrScenesStreetLampsLevels[bySceneID, 3];
		fbBACnet_AV_SL_Level_4.fPV  := GVL_IO.arrScenesStreetLampsLevels[bySceneID, 4];
		fbBACnet_AV_SL_Level_5.fPV  := GVL_IO.arrScenesStreetLampsLevels[bySceneID, 5];
		fbBACnet_AV_SL_Level_6.fPV  := GVL_IO.arrScenesStreetLampsLevels[bySceneID, 6];
		fbBACnet_AV_SL_Level_7.fPV  := GVL_IO.arrScenesStreetLampsLevels[bySceneID, 7];
		fbBACnet_AV_SL_Level_8.fPV  := GVL_IO.arrScenesStreetLampsLevels[bySceneID, 8];
		fbBACnet_AV_SL_Level_9.fPV  := GVL_IO.arrScenesStreetLampsLevels[bySceneID, 9];
		fbBACnet_AV_SL_Level_10.fPV := GVL_IO.arrScenesStreetLampsLevels[bySceneID, 10];
			
		iSelector := 0;		//after rewriting data go back to idle
		bBusy := FALSE;		//indicate that this FB is no longer busy
		
		
	128..254:	//SaveScene
		bBusy := TRUE;	//set a flag indicating that this FB is busy
		
		bySceneID := INT_TO_BYTE(iSelector) - 127;
		
		//iterate through arrays to
		FOR iCounter := 1 TO byStreetLampsCount BY 1 DO
			//save current lamp's power levels to memory buffer
			GVL_IO.arrScenesStreetLampsLevels[bySceneID, iCounter]
				:= GVL_IO.arrStreetLamps[iCounter].nLevel;
		END_FOR
		
		iSelector := 0;		//after saving data go back to idle
		bBusy := FALSE;		//indicate that this FB is no longer busy
		
END_CASE

END_FUNCTION_BLOCK

// ---- POUs/FB_PBL.TcPOU
FUNCTION_BLOCK FB_PBL
VAR_INPUT
	bSave		: BOOL;	// when rising edge occures, save current street lamp levels to arr_byPBL
	bRetrieve	: BOOL; // when rising edge occures, retrieve lamp levels from arr_byPBL
END_VAR
VAR_OUTPUT
END_VAR
VAR
	rtSave		: R_TRIG; // detects rising edge on bSave
	rtRetrieve	: R_TRIG; // detects rising edge on bRetrieve
	
	i			: INT;	// for loop iterator
	arr_byPBL	: ARRAY [1..byStreetLampsCount] OF BYTE;	// array of previous brightness levels
END_VAR

//init rising edge detection
rtSave(CLK := bSave);
rtRetrieve(CLK := bRetrieve);

//if rising edge occures on bSave
IF rtSave.Q THEN
	//iterate through street lamps and
	FOR i := 1 TO byStreetLampsCount BY 1 DO
		//save actual brightness levels to arr_byPBL
		arr_byPBL[i] := GVL_IO.arrStreetLamps[i].nLevel;
	END_FOR	
END_IF

//if rising edge occures on bRetrieve
IF rtRetrieve.Q THEN
	//retrive data from arr_byPBL and set lamps to those levels
	fbBACnet_AV_SL_Level_1.fPV  := arr_byPBL[1];
    fbBACnet_AV_SL_Level_2.fPV  := arr_byPBL[2];
    fbBACnet_AV_SL_Level_3.fPV  := arr_byPBL[3];
    fbBACnet_AV_SL_Level_4.fPV  := arr_byPBL[4];
    fbBACnet_AV_SL_Level_5.fPV  := arr_byPBL[5];
    fbBACnet_AV_SL_Level_6.fPV  := arr_byPBL[6];
    fbBACnet_AV_SL_Level_7.fPV  := arr_byPBL[7];
    fbBACnet_AV_SL_Level_8.fPV  := arr_byPBL[8];
    fbBACnet_AV_SL_Level_9.fPV  := arr_byPBL[9];
    fbBACnet_AV_SL_Level_10.fPV := arr_byPBL[10];
END_IF

END_FUNCTION_BLOCK

// ---- POUs/P_AddrAssignment.TcPOU
PROGRAM P_AddrAssignment
VAR
	iDoItOnceCounter	: INT := 0;
END_VAR

CASE iDoItOnceCounter OF
	0: // first cycle after download - assign addresses
		
		GVL_IO.arrStreetLamps[1].eKL6821Module  	:= eKL6821Module_none;
		GVL_IO.arrStreetLamps[1].nAddrShort1		:= 63;
		GVL_IO.arrStreetLamps[1].nAddrShort2		:= 63;
		                                        	
		GVL_IO.arrStreetLamps[2].eKL6821Module  	:= eKL6821Module_RB1;
		GVL_IO.arrStreetLamps[2].nAddrShort1		:= 2;
		GVL_IO.arrStreetLamps[2].nAddrShort2		:= 3;
		                                        	
		GVL_IO.arrStreetLamps[3].eKL6821Module  	:= eKL6821Module_RB1;
		GVL_IO.arrStreetLamps[3].nAddrShort1		:= 0;
		GVL_IO.arrStreetLamps[3].nAddrShort2		:= 1;
		                                        	
		GVL_IO.arrStreetLamps[4].eKL6821Module  	:= eKL6821Module_RB2;
		GVL_IO.arrStreetLamps[4].nAddrShort1		:= 0;
		GVL_IO.arrStreetLamps[4].nAddrShort2		:= 1;
		                                        	
		GVL_IO.arrStreetLamps[5].eKL6821Module  	:= eKL6821Module_RB2;
		GVL_IO.arrStreetLamps[5].nAddrShort1		:= 6;
		GVL_IO.arrStreetLamps[5].nAddrShort2		:= 7;
		                                        	
		GVL_IO.arrStreetLamps[6].eKL6821Module  	:= eKL6821Module_RB2;
		GVL_IO.arrStreetLamps[6].nAddrShort1		:= 3;
		GVL_IO.arrStreetLamps[6].nAddrShort2		:= 5;
		                                        	
		GVL_IO.arrStreetLamps[7].eKL6821Module  	:= eKL6821Module_RB2;
		GVL_IO.arrStreetLamps[7].nAddrShort1		:= 2;
		GVL_IO.arrStreetLamps[7].nAddrShort2		:= 4;
		                                        	
		GVL_IO.arrStreetLamps[8].eKL6821Module  	:= eKL6821Module_RB3;
		GVL_IO.arrStreetLamps[8].nAddrShort1		:= 0;
		GVL_IO.arrStreetLamps[8].nAddrShort2		:= 3;
		                                        	
		GVL_IO.arrStreetLamps[9].eKL6821Module  	:= eKL6821Module_RB3;
		GVL_IO.arrStreetLamps[9].nAddrShort1		:= 1;
		GVL_IO.arrStreetLamps[9].nAddrShort2		:= 2;
		                                        	
		GVL_IO.arrStreetLamps[10].eKL6821Module 	:= eKL6821Module_RB3;
		GVL_IO.arrStreetLamps[10].nAddrShort1		:= 4;
		GVL_IO.arrStreetLamps[10].nAddrShort2		:= 5;
		
		//increment to go to the next step wich is idle
		iDoItOnceCounter := iDoItOnceCounter + 1;
	
	1: // idle state
		; // do nothing
		
END_CASE

END_PROGRAM

// ---- POUs/KNX/P_MotionSensors.TcPOU
PROGRAM P_MotionSensors
VAR_INPUT
	bEnable		: BOOL; // if TRUE, program is active, sensors are taken into account
END_VAR
VAR
	i			: INT := 0;	// for loop iterator
	j			: INT := 0; // for loop iterator
	
	arrTOF_info	: ARRAY [1..byStreetLampsCount] OF TOF; 	// array of off-delay timers for short movement capture
	
	arrTOF		: ARRAY [1..byStreetLampsCount] OF TOF; 	// array of off-delay timers
	arrR_TRIG	: ARRAY [1..byStreetLampsCount] OF R_TRIG;	// array of rising edge trigers
	arrF_TRIG	: ARRAY [1..byStreetLampsCount] OF F_TRIG; 	// array of falling edge trigers
	
END_VAR

//time independent info about motion sensors
//iterate through street lamps
FOR j := 1 TO byStreetLampsCount BY 1 DO
	//initializing off-delay timers
	arrTOF_info[j](IN := GVL_IO.arrStreetLamps[j].bMotionSensor, PT := tMotionSensorsTOF_info_PT);
	//send motion info to ST
	GVL_IO.arrStreetLamps[j].bMotionFlag := arrTOF_info[j].Q;
END_FOR

//if motion sensors are activated and it is a night
IF bEnable AND F_IsNight() THEN
	
	//iterate through street lamps
	FOR i := 1 TO byStreetLampsCount BY 1 DO
		//if lamp is not in manual mode then
		IF NOT GVL_IO.arrStreetLamps[i].bManualCtrl THEN
			
			//start timers and edge detection
			//initializing off-delay timers
			arrTOF[i](IN := GVL_IO.arrStreetLamps[i].bMotionSensor, PT := tMotionSensorsTOF_PT);
			//initializing rising edge trigers
			arrR_TRIG[i](CLK := arrTOF[i].Q);
			//initializing falling edge trigers
			arrF_TRIG[i](CLK := arrTOF[i].Q);
			
			//if rising edge at arrTOF output occured
			IF arrR_TRIG[i].Q THEN
				//depending on a lamp, the sensor belongs to
				CASE i OF
					//turn the lamp in c_byBrightness_Motion mode
					1: fbBACnet_AV_SL_Level_1.fPV  := c_byBrightness_Motion;
					2: fbBACnet_AV_SL_Level_2.fPV  := c_byBrightness_Motion;
					3: fbBACnet_AV_SL_Level_3.fPV  := c_byBrightness_Motion;
					4: fbBACnet_AV_SL_Level_4.fPV  := c_byBrightness_Motion;
					5: fbBACnet_AV_SL_Level_5.fPV  := c_byBrightness_Motion;
					6: fbBACnet_AV_SL_Level_6.fPV  := c_byBrightness_Motion;
					7: fbBACnet_AV_SL_Level_7.fPV  := c_byBrightness_Motion;
					8: fbBACnet_AV_SL_Level_8.fPV  := c_byBrightness_Motion;
					9: fbBACnet_AV_SL_Level_9.fPV  := c_byBrightness_Motion;
					10:fbBACnet_AV_SL_Level_10.fPV := c_byBrightness_Motion;
				END_CASE
			//else if a falling edge at arrTOF output occured
			ELSIF arrF_TRIG[i].Q THEN
				//depending on a lamp, the sensor belongs to
				CASE i OF
					//turn the lamp in c_byBrightness_Night mode
					1: fbBACnet_AV_SL_Level_1.fPV  := c_byBrightness_Night;
					2: fbBACnet_AV_SL_Level_2.fPV  := c_byBrightness_Night;
					3: fbBACnet_AV_SL_Level_3.fPV  := c_byBrightness_Night;
					4: fbBACnet_AV_SL_Level_4.fPV  := c_byBrightness_Night;
					5: fbBACnet_AV_SL_Level_5.fPV  := c_byBrightness_Night;
					6: fbBACnet_AV_SL_Level_6.fPV  := c_byBrightness_Night;
					7: fbBACnet_AV_SL_Level_7.fPV  := c_byBrightness_Night;
					8: fbBACnet_AV_SL_Level_8.fPV  := c_byBrightness_Night;
					9: fbBACnet_AV_SL_Level_9.fPV  := c_byBrightness_Night;
					10:fbBACnet_AV_SL_Level_10.fPV := c_byBrightness_Night;
				END_CASE
			END_IF
		END_IF
	END_FOR
	
END_IF

END_PROGRAM

// ---- POUs/F_IsNight.TcPOU
FUNCTION F_IsNight : BOOL
VAR_INPUT
END_VAR
VAR
	fbCalcSunriseSunset 	: FB_CalcSunriseSunset;
	todSunrise          	: TOD;
	todSunset           	: TOD;
	fbGetSystemTime     	: GETSYSTEMTIME;
	fileTime            	: T_FILETIME;
	dtCurrentDateGMT		: DATE_AND_TIME;
	
	dtCurrentDate       	: DATE_AND_TIME;
	todCurrent				: TOD;
	
END_VAR

//get system time 
fbGetSystemTime(timeLoDW =>fileTime.dwLowDateTime, timeHiDW =>fileTime.dwHighDateTime);
dtCurrentDateGMT := FILETIME_TO_DT(fileTime);

//covert to UTC + 1
dtCurrentDate := dtCurrentDateGMT + T#1H;
todCurrent := DT_TO_TOD(dtCurrentDate);

//calculating sunrise and sunset
fbCalcSunriseSunset( fDegreeOfLongitude := 17.03,   (* Longitude of Wroclaw *)
					 fDegreeOfLatitude := 51.1,   (* Latitude of Wroclaw *)
					 fReferenceMeridian := 15.0,  (* Central European Time *)
					 dCurrentDate := DT_TO_DATE(dtCurrentDate),
					 todSunrise => todSunrise,
					 todSunset => todSunset);
							 
	
//if it is a night
IF todCurrent < todSunrise - T#1H OR todCurrent > todSunset THEN
	//set return value to TRUE
	F_IsNight := TRUE;
//else it is a day
ELSE
	//set return value to FALSE
	F_IsNight := FALSE;
END_IF

END_FUNCTION

// ---- POUs/P_AlarmMode.TcPOU
PROGRAM P_AlarmMode
VAR
	rtAlarm		: R_TRIG;
	ftAlarm		: F_TRIG;
	
	fbPBL		: FB_PBL;
END_VAR

//init rising and falling edge detection
rtAlarm(CLK := fbBACnet_BV_Alarm.bPresentValue);
ftAlarm(CLK := fbBACnet_BV_Alarm.bPresentValue);

//if rising edge occured
IF rtAlarm.Q THEN
	//save present brightness levels
	fbPBL(bSave := TRUE);
	//reset executive input
	fbPBL(bSave := FALSE);
	
	//reset manual mode
	bBACnet_ResetManual := TRUE;
	
	//then set street lamp levels to c_byBrightness_Alarm level
	fbBACnet_AV_SL_Level_1.fPV  := c_byBrightness_Alarm;
	fbBACnet_AV_SL_Level_2.fPV  := c_byBrightness_Alarm;
	fbBACnet_AV_SL_Level_3.fPV  := c_byBrightness_Alarm;
	fbBACnet_AV_SL_Level_4.fPV  := c_byBrightness_Alarm;
	fbBACnet_AV_SL_Level_5.fPV  := c_byBrightness_Alarm;
	fbBACnet_AV_SL_Level_6.fPV  := c_byBrightness_Alarm;
	fbBACnet_AV_SL_Level_7.fPV  := c_byBrightness_Alarm;
	fbBACnet_AV_SL_Level_8.fPV  := c_byBrightness_Alarm;
	fbBACnet_AV_SL_Level_9.fPV  := c_byBrightness_Alarm;
	fbBACnet_AV_SL_Level_10.fPV := c_byBrightness_Alarm;
	
END_IF

//if falling edge occured
IF ftAlarm.Q THEN
	//retrieve present brightness levels from memory
	fbPBL(bRetrieve := TRUE);
	//reset executive input
	fbPBL(bRetrieve := FALSE);
END_IF

END_PROGRAM

// ---- POUs/P_AutoMode.TcPOU
PROGRAM P_AutoMode
VAR
	tonCycle				: TON; //timer implemented to reduce CPU usage
	
	bIsDay			: BOOL := FALSE;
	bIsNight		: BOOL := FALSE;
	
	rtIsDay			: R_TRIG;
	rtIsNight		: R_TRIG;			
	
	ft_arrManual	: ARRAY [1..byStreetLampsCount] OF F_TRIG;
	i				: INT;	//for loop iterator
END_VAR

//init tonCycle
tonCycle(IN:=NOT tonCycle.Q, PT:=T#1S);
//init rising edge detection
rtIsDay(CLK := bIsDay);
rtIsNight(CLK := bIsNight);

//check day-night status every 1S
IF tonCycle.Q THEN
	
	//if it is a night
	IF F_IsNight() THEN
		//set flags accordingly
		bIsNight := TRUE;
		bIsDay := FALSE;
	//else, it is a day
	ELSE
		//set flags accordingly
		bIsNight := FALSE;
		bIsDay := TRUE;
	END_IF

END_IF

//if a night has come
IF rtIsNight.Q THEN
	//turn lights ON
	//if they are not in manual mode	
	IF NOT GVL_IO.arrStreetLamps[1].bManualCtrl  THEN fbBACnet_AV_SL_Level_1.fPV  := c_byBrightness_Night; END_IF
	IF NOT GVL_IO.arrStreetLamps[2].bManualCtrl  THEN fbBACnet_AV_SL_Level_2.fPV  := c_byBrightness_Night; END_IF
	IF NOT GVL_IO.arrStreetLamps[3].bManualCtrl  THEN fbBACnet_AV_SL_Level_3.fPV  := c_byBrightness_Night; END_IF
	IF NOT GVL_IO.arrStreetLamps[4].bManualCtrl  THEN fbBACnet_AV_SL_Level_4.fPV  := c_byBrightness_Night; END_IF
	IF NOT GVL_IO.arrStreetLamps[5].bManualCtrl  THEN fbBACnet_AV_SL_Level_5.fPV  := c_byBrightness_Night; END_IF
	IF NOT GVL_IO.arrStreetLamps[6].bManualCtrl  THEN fbBACnet_AV_SL_Level_6.fPV  := c_byBrightness_Night; END_IF
	IF NOT GVL_IO.arrStreetLamps[7].bManualCtrl  THEN fbBACnet_AV_SL_Level_7.fPV  := c_byBrightness_Night; END_IF
	IF NOT GVL_IO.arrStreetLamps[8].bManualCtrl  THEN fbBACnet_AV_SL_Level_8.fPV  := c_byBrightness_Night; END_IF
	IF NOT GVL_IO.arrStreetLamps[9].bManualCtrl  THEN fbBACnet_AV_SL_Level_9.fPV  := c_byBrightness_Night; END_IF
	IF NOT GVL_IO.arrStreetLamps[10].bManualCtrl THEN fbBACnet_AV_SL_Level_10.fPV := c_byBrightness_Night; END_IF

	//turn one street lamp ON
	GVL_IO.bStreetLamp_DO1 := TRUE;
END_IF

//if a day has come
IF rtIsDay.Q THEN
	//turn all lights OFF
	fbBACnet_AV_SL_Level_1.fPV  := c_byBrightness_Day;
	fbBACnet_AV_SL_Level_2.fPV  := c_byBrightness_Day;
	fbBACnet_AV_SL_Level_3.fPV  := c_byBrightness_Day;
	fbBACnet_AV_SL_Level_4.fPV  := c_byBrightness_Day;
	fbBACnet_AV_SL_Level_5.fPV  := c_byBrightness_Day;
	fbBACnet_AV_SL_Level_6.fPV  := c_byBrightness_Day;
	fbBACnet_AV_SL_Level_7.fPV  := c_byBrightness_Day;
	fbBACnet_AV_SL_Level_8.fPV  := c_byBrightness_Day;
	fbBACnet_AV_SL_Level_9.fPV  := c_byBrightness_Day;
	fbBACnet_AV_SL_Level_10.fPV := c_byBrightness_Day;
	
	//turn one street lamp OFF
	GVL_IO.bStreetLamp_DO1 := FALSE;
	
	//and disable manual mode
	bBACnet_ResetManual := TRUE;
END_IF

//special case - exit manual mode
//when manual mode is turned off
//return brightness level to auto mode level 
FOR i := 1 TO byStreetLampsCount BY 1 DO
	//init falling edge detection
	ft_arrManual[i](CLK := GVL_IO.arrStreetLamps[i].bManualCtrl);
	
	//if manual mode is being turned off
	IF ft_arrManual[i].Q THEN
		//set brightness level to auto mode on this lamp
		//in the night to c_byBrightness_Night
		IF F_IsNight() THEN
			CASE i OF
				1: 	fbBACnet_AV_SL_Level_1.fPV  := c_byBrightness_Night;
				2: 	fbBACnet_AV_SL_Level_2.fPV  := c_byBrightness_Night;
				3: 	fbBACnet_AV_SL_Level_3.fPV  := c_byBrightness_Night;
				4: 	fbBACnet_AV_SL_Level_4.fPV  := c_byBrightness_Night;
				5: 	fbBACnet_AV_SL_Level_5.fPV  := c_byBrightness_Night;
				6: 	fbBACnet_AV_SL_Level_6.fPV  := c_byBrightness_Night;
				7: 	fbBACnet_AV_SL_Level_7.fPV  := c_byBrightness_Night;
				8: 	fbBACnet_AV_SL_Level_8.fPV  := c_byBrightness_Night;
				9: 	fbBACnet_AV_SL_Level_9.fPV  := c_byBrightness_Night;
				10:	fbBACnet_AV_SL_Level_10.fPV := c_byBrightness_Night;
			END_CASE
		ELSE
		//at the daylight to c_byBrightness_Day
			CASE i OF
				1: 	fbBACnet_AV_SL_Level_1.fPV  := c_byBrightness_Day;
				2: 	fbBACnet_AV_SL_Level_2.fPV  := c_byBrightness_Day;
				3: 	fbBACnet_AV_SL_Level_3.fPV  := c_byBrightness_Day;
				4: 	fbBACnet_AV_SL_Level_4.fPV  := c_byBrightness_Day;
				5: 	fbBACnet_AV_SL_Level_5.fPV  := c_byBrightness_Day;
				6: 	fbBACnet_AV_SL_Level_6.fPV  := c_byBrightness_Day;
				7: 	fbBACnet_AV_SL_Level_7.fPV  := c_byBrightness_Day;
				8: 	fbBACnet_AV_SL_Level_8.fPV  := c_byBrightness_Day;
				9: 	fbBACnet_AV_SL_Level_9.fPV  := c_byBrightness_Day;
				10:	fbBACnet_AV_SL_Level_10.fPV := c_byBrightness_Day;
			END_CASE
		END_IF
	END_IF
END_FOR

END_PROGRAM

// ---- POUs/KNX/P_KNX_Data_MotionSensors.TcPOU
PROGRAM P_KNX_Data_MotionSensors
VAR
	EIB_BIT_REC_1		:EIB_BIT_REC;
	EIB_BIT_REC_2		:EIB_BIT_REC;
	EIB_BIT_REC_3		:EIB_BIT_REC;
	EIB_BIT_REC_4		:EIB_BIT_REC;
	EIB_BIT_REC_5		:EIB_BIT_REC;
	EIB_BIT_REC_6		:EIB_BIT_REC;
	EIB_BIT_REC_7		:EIB_BIT_REC;
	EIB_BIT_REC_8		:EIB_BIT_REC;
	EIB_BIT_REC_9		:EIB_BIT_REC;
	EIB_BIT_REC_10		:EIB_BIT_REC;
	EIB_BIT_REC_11		:EIB_BIT_REC;
	EIB_BIT_REC_12		:EIB_BIT_REC;
	EIB_BIT_REC_13		:EIB_BIT_REC;
	EIB_BIT_REC_14		:EIB_BIT_REC;
	EIB_BIT_REC_15		:EIB_BIT_REC;
	EIB_BIT_REC_16		:EIB_BIT_REC;
	
	Group_Address_1		: EIB_GROUP_ADDR := (MAIN := 12, SUB_MAIN := 0, NUMBER := 1);
	Group_Address_2		: EIB_GROUP_ADDR := (MAIN := 12, SUB_MAIN := 0, NUMBER := 2);
	Group_Address_3		: EIB_GROUP_ADDR := (MAIN := 12, SUB_MAIN := 0, NUMBER := 3);
	Group_Address_4		: EIB_GROUP_ADDR := (MAIN := 12, SUB_MAIN := 0, NUMBER := 4);
	Group_Address_5		: EIB_GROUP_ADDR := (MAIN := 12, SUB_MAIN := 0, NUMBER := 5);
	Group_Address_6		: EIB_GROUP_ADDR := (MAIN := 12, SUB_MAIN := 0, NUMBER := 6);
	Group_Address_7		: EIB_GROUP_ADDR := (MAIN := 12, SUB_MAIN := 0, NUMBER := 7);
	Group_Address_8		: EIB_GROUP_ADDR := (MAIN := 12, SUB_MAIN := 0, NUMBER := 8);
	Group_Address_9		: EIB_GROUP_ADDR := (MAIN := 12, SUB_MAIN := 0, NUMBER := 9);
	Group_Address_10	: EIB_GROUP_ADDR := (MAIN := 12, SUB_MAIN := 0, NUMBER := 10);
	Group_Address_11	: EIB_GROUP_ADDR := (MAIN := 12, SUB_MAIN := 0, NUMBER := 11);
	Group_Address_12	: EIB_GROUP_ADDR := (MAIN := 12, SUB_MAIN := 0, NUMBER := 12);
	Group_Address_13	: EIB_GROUP_ADDR := (MAIN := 12, SUB_MAIN := 0, NUMBER := 13);
	Group_Address_14	: EIB_GROUP_ADDR := (MAIN := 12, SUB_MAIN := 0, NUMBER := 14);
	Group_Address_15	: EIB_GROUP_ADDR := (MAIN := 12, SUB_MAIN := 0, NUMBER := 15);
	Group_Address_16	: EIB_GROUP_ADDR := (MAIN := 12, SUB_MAIN := 0, NUMBER := 16);
	
END_VAR

//EIB_BIT_REC function block initialization
EIB_BIT_REC_1(Group_Address:=Group_Address_1, strData_Rec:=GVL_IO.str_Data_Rec);
EIB_BIT_REC_2(Group_Address:=Group_Address_2, strData_Rec:=GVL_IO.str_Data_Rec);
EIB_BIT_REC_3(Group_Address:=Group_Address_3, strData_Rec:=GVL_IO.str_Data_Rec);
EIB_BIT_REC_4(Group_Address:=Group_Address_4, strData_Rec:=GVL_IO.str_Data_Rec);
EIB_BIT_REC_5(Group_Address:=Group_Address_5, strData_Rec:=GVL_IO.str_Data_Rec);
EIB_BIT_REC_6(Group_Address:=Group_Address_6, strData_Rec:=GVL_IO.str_Data_Rec);
EIB_BIT_REC_7(Group_Address:=Group_Address_7, strData_Rec:=GVL_IO.str_Data_Rec);
EIB_BIT_REC_8(Group_Address:=Group_Address_8, strData_Rec:=GVL_IO.str_Data_Rec);
EIB_BIT_REC_9(Group_Address:=Group_Address_9, strData_Rec:=GVL_IO.str_Data_Rec);
EIB_BIT_REC_10(Group_Address:=Group_Address_10, strData_Rec:=GVL_IO.str_Data_Rec);
EIB_BIT_REC_11(Group_Address:=Group_Address_11, strData_Rec:=GVL_IO.str_Data_Rec);
EIB_BIT_REC_12(Group_Address:=Group_Address_12, strData_Rec:=GVL_IO.str_Data_Rec);
EIB_BIT_REC_13(Group_Address:=Group_Address_13, strData_Rec:=GVL_IO.str_Data_Rec);
EIB_BIT_REC_14(Group_Address:=Group_Address_14, strData_Rec:=GVL_IO.str_Data_Rec);
EIB_BIT_REC_15(Group_Address:=Group_Address_15, strData_Rec:=GVL_IO.str_Data_Rec);
EIB_BIT_REC_16(Group_Address:=Group_Address_16, strData_Rec:=GVL_IO.str_Data_Rec);

//Assign value to lamp motion sensor variables
GVL_IO.arrStreetLamps[1].bMotionSensor := FALSE;
GVL_IO.arrStreetLamps[2].bMotionSensor := EIB_BIT_REC_1.bData OR EIB_BIT_REC_2.bData;
GVL_IO.arrStreetLamps[3].bMotionSensor := EIB_BIT_REC_3.bData OR EIB_BIT_REC_4.bData;
GVL_IO.arrStreetLamps[4].bMotionSensor := EIB_BIT_REC_5.bData OR EIB_BIT_REC_6.bData;
GVL_IO.arrStreetLamps[5].bMotionSensor := EIB_BIT_REC_11.bData;
GVL_IO.arrStreetLamps[6].bMotionSensor := EIB_BIT_REC_7.bData OR EIB_BIT_REC_8.bData;
GVL_IO.arrStreetLamps[7].bMotionSensor := EIB_BIT_REC_12.bData;
GVL_IO.arrStreetLamps[8].bMotionSensor := EIB_BIT_REC_13.bData OR EIB_BIT_REC_14.bData;
GVL_IO.arrStreetLamps[9].bMotionSensor := EIB_BIT_REC_15.bData OR EIB_BIT_REC_16.bData;
GVL_IO.arrStreetLamps[10].bMotionSensor := EIB_BIT_REC_9.bData OR EIB_BIT_REC_10.bData;

END_PROGRAM

// ---- POUs/KNX/P_KNX_Data_GatesANDAlarm.TcPOU
PROGRAM P_KNX_Data_GatesANDAlarm
VAR
	EIB_BIT_SEND_1		:EIB_BIT_SEND;
	EIB_BIT_SEND_2		:EIB_BIT_SEND;
	EIB_BIT_SEND_3		:EIB_BIT_SEND;
	EIB_BIT_SEND_4		:EIB_BIT_SEND;
	EIB_BIT_SEND_5		:EIB_BIT_SEND;
	EIB_BIT_SEND_6		:EIB_BIT_SEND;
	EIB_BIT_SEND_7		:EIB_BIT_SEND;
	EIB_BIT_SEND_8		:EIB_BIT_SEND;
	EIB_BIT_REC_9		:EIB_BIT_REC;
	
	Group_Address_1		: EIB_GROUP_ADDR := (MAIN := 12, SUB_MAIN := 1, NUMBER := 0);	//barrier
	Group_Address_2		: EIB_GROUP_ADDR := (MAIN := 12, SUB_MAIN := 1, NUMBER := 1);	//main gate
	Group_Address_3		: EIB_GROUP_ADDR := (MAIN := 12, SUB_MAIN := 1, NUMBER := 2);	//gateway and barrier
	Group_Address_4		: EIB_GROUP_ADDR := (MAIN := 12, SUB_MAIN := 1, NUMBER := 3);	//garage door
	Group_Address_5		: EIB_GROUP_ADDR := (MAIN := 12, SUB_MAIN := 1, NUMBER := 4);	//left curtain
	Group_Address_6		: EIB_GROUP_ADDR := (MAIN := 12, SUB_MAIN := 1, NUMBER := 5);	//right curtain
	Group_Address_7		: EIB_GROUP_ADDR := (MAIN := 12, SUB_MAIN := 1, NUMBER := 9);	//rear gate
	Group_Address_8		: EIB_GROUP_ADDR := (MAIN := 12, SUB_MAIN := 1, NUMBER := 10);	//rear gateway
	Group_Address_9		: EIB_GROUP_ADDR := (MAIN := 12, SUB_MAIN := 1, NUMBER := 37);	//intrusion alarm
	
	dwGates				: DWORD;
	rGates				: REAL;
END_VAR

//keep BACnet object instance alive
fbBACnet_AV_Gates(Device := Device);
//read gates values from BACnet object
rGates := fbBACnet_AV_Gates.fPresentValue;
//convert REAL to DWORD
dwGates := REAL_TO_DWORD(rGates);


//EIB_BIT_SEND function block initialization
//with data write from BACnet object
EIB_BIT_SEND_1(Group_Address:=Group_Address_1, bData := dwGates.0 , str_Rec:=GVL_IO.str_Data_Rec);
EIB_BIT_SEND_2(Group_Address:=Group_Address_2, bData := dwGates.1 , str_Rec:=GVL_IO.str_Data_Rec);
EIB_BIT_SEND_3(Group_Address:=Group_Address_3, bData := dwGates.2 , str_Rec:=GVL_IO.str_Data_Rec);
EIB_BIT_SEND_4(Group_Address:=Group_Address_4, bData := dwGates.3 , str_Rec:=GVL_IO.str_Data_Rec);
EIB_BIT_SEND_5(Group_Address:=Group_Address_5, bData := dwGates.4 , str_Rec:=GVL_IO.str_Data_Rec);
EIB_BIT_SEND_6(Group_Address:=Group_Address_6, bData := dwGates.5 , str_Rec:=GVL_IO.str_Data_Rec);
EIB_BIT_SEND_7(Group_Address:=Group_Address_7, bData := dwGates.6 , str_Rec:=GVL_IO.str_Data_Rec);
EIB_BIT_SEND_8(Group_Address:=Group_Address_8, bData := dwGates.7 , str_Rec:=GVL_IO.str_Data_Rec);
//EIB_BIT_REC function block initialization
EIB_BIT_REC_9(Group_Address:=Group_Address_9, strData_Rec:=GVL_IO.str_Data_Rec);


//keep BACnet object instance alive
//assign alarm value to BACnet object
fbBACnet_BV_Alarm(Device := Device, bEnablePV := TRUE, bNullPV := FALSE, bPV := EIB_BIT_REC_9.bData);

END_PROGRAM

// ---- POUs/DimmersStreetLamps/P_Dimmers_RB1.TcPOU
PROGRAM P_Dimmers_RB1
VAR
	fbDALIV2Dimmer2Switch_RB1_1		: FB_DALIV2Dimmer2Switch;
	nActualLEvelMasterDev_1			: BYTE;
	bBusy_1							: BOOL;
	bError_1						: BOOL;
	nErrorId_1						: UDINT;
	
	
	fbDALIV2Dimmer2Switch_RB1_2		: FB_DALIV2Dimmer2Switch;
	nActualLEvelMasterDev_2			: BYTE;
	bBusy_2							: BOOL;
	bError_2						: BOOL;
	nErrorId_2						: UDINT;
	
	
	fbDALIV2Dimmer2Switch_RB1_3		: FB_DALIV2Dimmer2Switch;
	nActualLEvelMasterDev_3			: BYTE;
	bBusy_3							: BOOL;
	bError_3						: BOOL;
	nErrorId_3						: UDINT;
	
	fbDALIV2Dimmer2Switch_RB1_4		: FB_DALIV2Dimmer2Switch;
	nActualLEvelMasterDev_4			: BYTE;
	bBusy_4							: BOOL;
	bError_4						: BOOL;
	nErrorId_4						: UDINT;
	
	fbDALIV2Dimmer2Switch_RB1_5		: FB_DALIV2Dimmer2Switch;
	nActualLEvelMasterDev_5			: BYTE;
	bBusy_5							: BOOL;
	bError_5						: BOOL;
	nErrorId_5						: UDINT;
	
	fbDALIV2Dimmer2Switch_RB1_6		: FB_DALIV2Dimmer2Switch;
	nActualLEvelMasterDev_6			: BYTE;
	bBusy_6							: BOOL;
	bError_6						: BOOL;
	nErrorId_6						: UDINT;

END_VAR

fbDALIV2Dimmer2Switch_RB1_2(
    bSetDimmValue := GVL_StreetLamps.bSetDimmValue,
    nDimmValue := GVL_IO.arrStreetLamps[1].nLevel,
    tSwitchOverTime := GVL_StreetLamps.tSwitchOverTime,
    bMemoryModeOn := GVL_StreetLamps.bMemoryModeOn,
    nOnValueWithoutMemoryMode := GVL_StreetLamps.nOnValueWithoutMemoryMode,
    nAddr := GVL_IO.arrStreetLamps[1].nAddrShort2,
    eAddrType := eDALIV2AddrTypeShort,
    nMasterDevAddr := GVL_StreetLamps.nMasterDevAddr,
    tCycleActualLevelMasterDev := GVL_StreetLamps.tCycleActualLevelMasterDev,
    stCommandBuffer := GVL_IO.stCommandBuffer_RB1); // FB_DALIV2Dimmer2Switch
fbDALIV2Dimmer2Switch_RB1_1(
    bSetDimmValue := GVL_StreetLamps.bSetDimmValue,
    nDimmValue := GVL_IO.arrStreetLamps[1].nLevel,
    tSwitchOverTime := GVL_StreetLamps.tSwitchOverTime,
    bMemoryModeOn := GVL_StreetLamps.bMemoryModeOn,
    nOnValueWithoutMemoryMode := GVL_StreetLamps.nOnValueWithoutMemoryMode,
    nAddr := GVL_IO.arrStreetLamps[1].nAddrShort1,
    eAddrType := eDALIV2AddrTypeShort,
    nMasterDevAddr := GVL_StreetLamps.nMasterDevAddr,
    tCycleActualLevelMasterDev := GVL_StreetLamps.tCycleActualLevelMasterDev,
    stCommandBuffer := GVL_IO.stCommandBuffer_RB1); // FB_DALIV2Dimmer2Switch
nActualLEvelMasterDev_2 := fbDALIV2Dimmer2Switch_RB1_2.nActualLevelMasterDev;
fbDALIV2Dimmer2Switch_RB1_3(
    bSetDimmValue := GVL_StreetLamps.bSetDimmValue,
    nDimmValue := GVL_IO.arrStreetLamps[2].nLevel,
    tSwitchOverTime := GVL_StreetLamps.tSwitchOverTime,
    bMemoryModeOn := GVL_StreetLamps.bMemoryModeOn,
    nOnValueWithoutMemoryMode := GVL_StreetLamps.nOnValueWithoutMemoryMode,
    nAddr := GVL_IO.arrStreetLamps[2].nAddrShort1,
    eAddrType := eDALIV2AddrTypeShort,
    nMasterDevAddr := GVL_StreetLamps.nMasterDevAddr,
    tCycleActualLevelMasterDev := GVL_StreetLamps.tCycleActualLevelMasterDev,
    stCommandBuffer := GVL_IO.stCommandBuffer_RB1); // FB_DALIV2Dimmer2Switch
bBusy_2 := fbDALIV2Dimmer2Switch_RB1_2.bBusy;
nActualLEvelMasterDev_1 := fbDALIV2Dimmer2Switch_RB1_1.nActualLevelMasterDev;
bBusy_1 := fbDALIV2Dimmer2Switch_RB1_1.bBusy;
bError_2 := fbDALIV2Dimmer2Switch_RB1_2.bError;
bError_1 := fbDALIV2Dimmer2Switch_RB1_1.bError;
nErrorId_2 := fbDALIV2Dimmer2Switch_RB1_2.nErrorId;
nActualLEvelMasterDev_3 := fbDALIV2Dimmer2Switch_RB1_3.nActualLevelMasterDev;
bBusy_3 := fbDALIV2Dimmer2Switch_RB1_3.bBusy;
nErrorId_1 := fbDALIV2Dimmer2Switch_RB1_1.nErrorId;
bError_3 := fbDALIV2Dimmer2Switch_RB1_3.bError;
nErrorId_3 := fbDALIV2Dimmer2Switch_RB1_3.nErrorId;
fbDALIV2Dimmer2Switch_RB1_4(
    bSetDimmValue := GVL_StreetLamps.bSetDimmValue,
    nDimmValue := GVL_IO.arrStreetLamps[2].nLevel,
    tSwitchOverTime := GVL_StreetLamps.tSwitchOverTime,
    bMemoryModeOn := GVL_StreetLamps.bMemoryModeOn,
    nOnValueWithoutMemoryMode := GVL_StreetLamps.nOnValueWithoutMemoryMode,
    nAddr := GVL_IO.arrStreetLamps[2].nAddrShort2,
    eAddrType := eDALIV2AddrTypeShort,
    nMasterDevAddr := GVL_StreetLamps.nMasterDevAddr,
    tCycleActualLevelMasterDev := GVL_StreetLamps.tCycleActualLevelMasterDev,
    stCommandBuffer := GVL_IO.stCommandBuffer_RB1); // FB_DALIV2Dimmer2Switch
nActualLEvelMasterDev_4 := fbDALIV2Dimmer2Switch_RB1_4.nActualLevelMasterDev;
bBusy_4 := fbDALIV2Dimmer2Switch_RB1_4.bBusy;
bError_4 := fbDALIV2Dimmer2Switch_RB1_4.bError;
nErrorId_4 := fbDALIV2Dimmer2Switch_RB1_4.nErrorId;
fbDALIV2Dimmer2Switch_RB1_5(
    bSetDimmValue := GVL_StreetLamps.bSetDimmValue,
    nDimmValue := GVL_IO.arrStreetLamps[3].nLevel,
    tSwitchOverTime := GVL_StreetLamps.tSwitchOverTime,
    bMemoryModeOn := GVL_StreetLamps.bMemoryModeOn,
    nOnValueWithoutMemoryMode := GVL_StreetLamps.nOnValueWithoutMemoryMode,
    nAddr := GVL_IO.arrStreetLamps[3].nAddrShort1,
    eAddrType := eDALIV2AddrTypeShort,
    nMasterDevAddr := GVL_StreetLamps.nMasterDevAddr,
    tCycleActualLevelMasterDev := GVL_StreetLamps.tCycleActualLevelMasterDev,
    stCommandBuffer := GVL_IO.stCommandBuffer_RB1); // FB_DALIV2Dimmer2Switch
nActualLEvelMasterDev_5 := fbDALIV2Dimmer2Switch_RB1_5.nActualLevelMasterDev;
bBusy_5 := fbDALIV2Dimmer2Switch_RB1_5.bBusy;
bError_5 := fbDALIV2Dimmer2Switch_RB1_5.bError;
nErrorId_5 := fbDALIV2Dimmer2Switch_RB1_5.nErrorId;
fbDALIV2Dimmer2Switch_RB1_6(
    bSetDimmValue := GVL_StreetLamps.bSetDimmValue,
    nDimmValue := GVL_IO.arrStreetLamps[3].nLevel,
    tSwitchOverTime := GVL_StreetLamps.tSwitchOverTime,
    bMemoryModeOn := GVL_StreetLamps.bMemoryModeOn,
    nOnValueWithoutMemoryMode := GVL_StreetLamps.nOnValueWithoutMemoryMode,
    nAddr := GVL_IO.arrStreetLamps[3].nAddrShort2,
    eAddrType := eDALIV2AddrTypeShort,
    nMasterDevAddr := GVL_StreetLamps.nMasterDevAddr,
    tCycleActualLevelMasterDev := GVL_StreetLamps.tCycleActualLevelMasterDev,
    stCommandBuffer := GVL_IO.stCommandBuffer_RB1); // FB_DALIV2Dimmer2Switch
nActualLEvelMasterDev_6 := fbDALIV2Dimmer2Switch_RB1_6.nActualLevelMasterDev;
bBusy_6 := fbDALIV2Dimmer2Switch_RB1_6.bBusy;
bError_6 := fbDALIV2Dimmer2Switch_RB1_6.bError;
nErrorId_6 := fbDALIV2Dimmer2Switch_RB1_6.nErrorId;

END_PROGRAM

// ---- POUs/DimmersStreetLamps/P_Dimmers_RB2.TcPOU
PROGRAM P_Dimmers_RB2
VAR
	fbDALIV2Dimmer2Switch_RB2_1		: FB_DALIV2Dimmer2Switch;
	nActualLEvelMasterDev_1			: BYTE;
	bBusy_1							: BOOL;
	bError_1						: BOOL;
	nErrorId_1						: UDINT;
	
	
	fbDALIV2Dimmer2Switch_RB2_2		: FB_DALIV2Dimmer2Switch;
	nActualLEvelMasterDev_2			: BYTE;
	bBusy_2							: BOOL;
	bError_2						: BOOL;
	nErrorId_2						: UDINT;
	
	
	fbDALIV2Dimmer2Switch_RB2_3		: FB_DALIV2Dimmer2Switch;
	nActualLEvelMasterDev_3			: BYTE;
	bBusy_3							: BOOL;
	bError_3						: BOOL;
	nErrorId_3						: UDINT;
	
	fbDALIV2Dimmer2Switch_RB2_4		: FB_DALIV2Dimmer2Switch;
	nActualLEvelMasterDev_4			: BYTE;
	bBusy_4							: BOOL;
	bError_4						: BOOL;
	nErrorId_4						: UDINT;
	
	fbDALIV2Dimmer2Switch_RB2_5		: FB_DALIV2Dimmer2Switch;
	nActualLEvelMasterDev_5			: BYTE;
	bBusy_5							: BOOL;
	bError_5						: BOOL;
	nErrorId_5						: UDINT;
	
	fbDALIV2Dimmer2Switch_RB2_6		: FB_DALIV2Dimmer2Switch;
	nActualLEvelMasterDev_6			: BYTE;
	bBusy_6							: BOOL;
	bError_6						: BOOL;
	nErrorId_6						: UDINT;
	
	fbDALIV2Dimmer2Switch_RB2_7		: FB_DALIV2Dimmer2Switch;
	nActualLEvelMasterDev_7			: BYTE;
	bBusy_7							: BOOL;
	bError_7						: BOOL;
	nErrorId_7						: UDINT;
	
	fbDALIV2Dimmer2Switch_RB2_8		: FB_DALIV2Dimmer2Switch;
	nActualLEvelMasterDev_8			: BYTE;
	bBusy_8							: BOOL;
	bError_8						: BOOL;
	nErrorId_8						: UDINT;
	
END_VAR

fbDALIV2Dimmer2Switch_RB2_2(
    bSetDimmValue := GVL_StreetLamps.bSetDimmValue,
    nDimmValue := GVL_IO.arrStreetLamps[5].nLevel,
    tSwitchOverTime := GVL_StreetLamps.tSwitchOverTime,
    bMemoryModeOn := GVL_StreetLamps.bMemoryModeOn,
    nOnValueWithoutMemoryMode := GVL_StreetLamps.nOnValueWithoutMemoryMode,
    nAddr := GVL_IO.arrStreetLamps[5].nAddrShort2,
    eAddrType := eDALIV2AddrTypeShort,
    nMasterDevAddr := GVL_StreetLamps.nMasterDevAddr,
    tCycleActualLevelMasterDev := GVL_StreetLamps.tCycleActualLevelMasterDev,
    stCommandBuffer := GVL_IO.stCommandBuffer_RB2); // FB_DALIV2Dimmer2Switch
fbDALIV2Dimmer2Switch_RB2_1(
    bSetDimmValue := GVL_StreetLamps.bSetDimmValue,
    nDimmValue := GVL_IO.arrStreetLamps[5].nLevel,
    tSwitchOverTime := GVL_StreetLamps.tSwitchOverTime,
    bMemoryModeOn := GVL_StreetLamps.bMemoryModeOn,
    nOnValueWithoutMemoryMode := GVL_StreetLamps.nOnValueWithoutMemoryMode,
    nAddr := GVL_IO.arrStreetLamps[5].nAddrShort1,
    eAddrType := eDALIV2AddrTypeShort,
    nMasterDevAddr := GVL_StreetLamps.nMasterDevAddr,
    tCycleActualLevelMasterDev := GVL_StreetLamps.tCycleActualLevelMasterDev,
    stCommandBuffer := GVL_IO.stCommandBuffer_RB2); // FB_DALIV2Dimmer2Switch
nActualLEvelMasterDev_2 := fbDALIV2Dimmer2Switch_RB2_2.nActualLevelMasterDev;
fbDALIV2Dimmer2Switch_RB2_3(
    bSetDimmValue := GVL_StreetLamps.bSetDimmValue,
    nDimmValue := GVL_IO.arrStreetLamps[6].nLevel,
    tSwitchOverTime := GVL_StreetLamps.tSwitchOverTime,
    bMemoryModeOn := GVL_StreetLamps.bMemoryModeOn,
    nOnValueWithoutMemoryMode := GVL_StreetLamps.nOnValueWithoutMemoryMode,
    nAddr := GVL_IO.arrStreetLamps[6].nAddrShort1,
    eAddrType := eDALIV2AddrTypeShort,
    nMasterDevAddr := GVL_StreetLamps.nMasterDevAddr,
    tCycleActualLevelMasterDev := GVL_StreetLamps.tCycleActualLevelMasterDev,
    stCommandBuffer := GVL_IO.stCommandBuffer_RB2); // FB_DALIV2Dimmer2Switch
bBusy_2 := fbDALIV2Dimmer2Switch_RB2_2.bBusy;
nActualLEvelMasterDev_1 := fbDALIV2Dimmer2Switch_RB2_1.nActualLevelMasterDev;
bBusy_1 := fbDALIV2Dimmer2Switch_RB2_1.bBusy;
bError_2 := fbDALIV2Dimmer2Switch_RB2_2.bError;
bError_1 := fbDALIV2Dimmer2Switch_RB2_1.bError;
nErrorId_2 := fbDALIV2Dimmer2Switch_RB2_2.nErrorId;
nActualLEvelMasterDev_3 := fbDALIV2Dimmer2Switch_RB2_3.nActualLevelMasterDev;
bBusy_3 := fbDALIV2Dimmer2Switch_RB2_3.bBusy;
nErrorId_1 := fbDALIV2Dimmer2Switch_RB2_1.nErrorId;
bError_3 := fbDALIV2Dimmer2Switch_RB2_3.bError;
nErrorId_3 := fbDALIV2Dimmer2Switch_RB2_3.nErrorId;
fbDALIV2Dimmer2Switch_RB2_4(
    bSetDimmValue := GVL_StreetLamps.bSetDimmValue,
    nDimmValue := GVL_IO.arrStreetLamps[6].nLevel,
    tSwitchOverTime := GVL_StreetLamps.tSwitchOverTime,
    bMemoryModeOn := GVL_StreetLamps.bMemoryModeOn,
    nOnValueWithoutMemoryMode := GVL_StreetLamps.nOnValueWithoutMemoryMode,
    nAddr := GVL_IO.arrStreetLamps[6].nAddrShort2,
    eAddrType := eDALIV2AddrTypeShort,
    nMasterDevAddr := GVL_StreetLamps.nMasterDevAddr,
    tCycleActualLevelMasterDev := GVL_StreetLamps.tCycleActualLevelMasterDev,
    stCommandBuffer := GVL_IO.stCommandBuffer_RB2); // FB_DALIV2Dimmer2Switch
nActualLEvelMasterDev_4 := fbDALIV2Dimmer2Switch_RB2_4.nActualLevelMasterDev;
bBusy_4 := fbDALIV2Dimmer2Switch_RB2_4.bBusy;
bError_4 := fbDALIV2Dimmer2Switch_RB2_4.bError;
nErrorId_4 := fbDALIV2Dimmer2Switch_RB2_4.nErrorId;
fbDALIV2Dimmer2Switch_RB2_5(
    bSetDimmValue := GVL_StreetLamps.bSetDimmValue,
    nDimmValue := GVL_IO.arrStreetLamps[7].nLevel,
    tSwitchOverTime := GVL_StreetLamps.tSwitchOverTime,
    bMemoryModeOn := GVL_StreetLamps.bMemoryModeOn,
    nOnValueWithoutMemoryMode := GVL_StreetLamps.nOnValueWithoutMemoryMode,
    nAddr := GVL_IO.arrStreetLamps[7].nAddrShort1,
    eAddrType := eDALIV2AddrTypeShort,
    nMasterDevAddr := GVL_StreetLamps.nMasterDevAddr,
    tCycleActualLevelMasterDev := GVL_StreetLamps.tCycleActualLevelMasterDev,
    stCommandBuffer := GVL_IO.stCommandBuffer_RB2); // FB_DALIV2Dimmer2Switch
nActualLEvelMasterDev_5 := fbDALIV2Dimmer2Switch_RB2_5.nActualLevelMasterDev;
bBusy_5 := fbDALIV2Dimmer2Switch_RB2_5.bBusy;
bError_5 := fbDALIV2Dimmer2Switch_RB2_5.bError;
nErrorId_5 := fbDALIV2Dimmer2Switch_RB2_5.nErrorId;
fbDALIV2Dimmer2Switch_RB2_6(
    bSetDimmValue := GVL_StreetLamps.bSetDimmValue,
    nDimmValue := GVL_IO.arrStreetLamps[7].nLevel,
    tSwitchOverTime := GVL_StreetLamps.tSwitchOverTime,
    bMemoryModeOn := GVL_StreetLamps.bMemoryModeOn,
    nOnValueWithoutMemoryMode := GVL_StreetLamps.nOnValueWithoutMemoryMode,
    nAddr := GVL_IO.arrStreetLamps[7].nAddrShort2,
    eAddrType := eDALIV2AddrTypeShort,
    nMasterDevAddr := GVL_StreetLamps.nMasterDevAddr,
    tCycleActualLevelMasterDev := GVL_StreetLamps.tCycleActualLevelMasterDev,
    stCommandBuffer := GVL_IO.stCommandBuffer_RB2); // FB_DALIV2Dimmer2Switch
nActualLEvelMasterDev_6 := fbDALIV2Dimmer2Switch_RB2_6.nActualLevelMasterDev;
bBusy_6 := fbDALIV2Dimmer2Switch_RB2_6.bBusy;
bError_6 := fbDALIV2Dimmer2Switch_RB2_6.bError;
nErrorId_6 := fbDALIV2Dimmer2Switch_RB2_6.nErrorId;
fbDALIV2Dimmer2Switch_RB2_7(
    bSetDimmValue := GVL_StreetLamps.bSetDimmValue,
    nDimmValue := GVL_IO.arrStreetLamps[4].nLevel,
    tSwitchOverTime := GVL_StreetLamps.tSwitchOverTime,
    bMemoryModeOn := GVL_StreetLamps.bMemoryModeOn,
    nOnValueWithoutMemoryMode := GVL_StreetLamps.nOnValueWithoutMemoryMode,
    nAddr := GVL_IO.arrStreetLamps[4].nAddrShort1,
    eAddrType := eDALIV2AddrTypeShort,
    nMasterDevAddr := GVL_StreetLamps.nMasterDevAddr,
    tCycleActualLevelMasterDev := GVL_StreetLamps.tCycleActualLevelMasterDev,
    stCommandBuffer := GVL_IO.stCommandBuffer_RB2); // FB_DALIV2Dimmer2Switch
nActualLEvelMasterDev_7 := fbDALIV2Dimmer2Switch_RB2_7.nActualLevelMasterDev;
bBusy_7 := fbDALIV2Dimmer2Switch_RB2_7.bBusy;
bError_7 := fbDALIV2Dimmer2Switch_RB2_7.bError;
nErrorId_7 := fbDALIV2Dimmer2Switch_RB2_7.nErrorId;
fbDALIV2Dimmer2Switch_RB2_8(
    bSetDimmValue := GVL_StreetLamps.bSetDimmValue,
    nDimmValue := GVL_IO.arrStreetLamps[4].nLevel,
    tSwitchOverTime := GVL_StreetLamps.tSwitchOverTime,
    bMemoryModeOn := GVL_StreetLamps.bMemoryModeOn,
    nOnValueWithoutMemoryMode := GVL_StreetLamps.nOnValueWithoutMemoryMode,
    nAddr := GVL_IO.arrStreetLamps[4].nAddrShort2,
    eAddrType := eDALIV2AddrTypeShort,
    nMasterDevAddr := GVL_StreetLamps.nMasterDevAddr,
    tCycleActualLevelMasterDev := GVL_StreetLamps.tCycleActualLevelMasterDev,
    stCommandBuffer := GVL_IO.stCommandBuffer_RB2); // FB_DALIV2Dimmer2Switch
nActualLEvelMasterDev_8 := fbDALIV2Dimmer2Switch_RB2_8.nActualLevelMasterDev;
bBusy_8 := fbDALIV2Dimmer2Switch_RB2_8.bBusy;
bError_8 := fbDALIV2Dimmer2Switch_RB2_8.bError;
nErrorId_8 := fbDALIV2Dimmer2Switch_RB2_8.nErrorId;

END_PROGRAM

// ---- POUs/DimmersStreetLamps/P_Dimmers_RB3.TcPOU
PROGRAM P_Dimmers_RB3
VAR
	fbDALIV2Dimmer2Switch_RB3_1		: FB_DALIV2Dimmer2Switch;
	nActualLEvelMasterDev_1			: BYTE;
	bBusy_1							: BOOL;
	bError_1						: BOOL;
	nErrorId_1						: UDINT;
	
	
	fbDALIV2Dimmer2Switch_RB3_2		: FB_DALIV2Dimmer2Switch;
	nActualLEvelMasterDev_2			: BYTE;
	bBusy_2							: BOOL;
	bError_2						: BOOL;
	nErrorId_2						: UDINT;
	
	
	fbDALIV2Dimmer2Switch_RB3_3		: FB_DALIV2Dimmer2Switch;
	nActualLEvelMasterDev_3			: BYTE;
	bBusy_3							: BOOL;
	bError_3						: BOOL;
	nErrorId_3						: UDINT;
	
	fbDALIV2Dimmer2Switch_RB3_4		: FB_DALIV2Dimmer2Switch;
	nActualLEvelMasterDev_4			: BYTE;
	bBusy_4							: BOOL;
	bError_4						: BOOL;
	nErrorId_4						: UDINT;
	
	fbDALIV2Dimmer2Switch_RB3_5		: FB_DALIV2Dimmer2Switch;
	nActualLEvelMasterDev_5			: BYTE;
	bBusy_5							: BOOL;
	bError_5						: BOOL;
	nErrorId_5						: UDINT;
	
	fbDALIV2Dimmer2Switch_RB3_6		: FB_DALIV2Dimmer2Switch;
	nActualLEvelMasterDev_6			: BYTE;
	bBusy_6							: BOOL;
	bError_6						: BOOL;
	nErrorId_6						: UDINT;
	
END_VAR

fbDALIV2Dimmer2Switch_RB3_2(
    bSetDimmValue := GVL_StreetLamps.bSetDimmValue,
    nDimmValue := GVL_IO.arrStreetLamps[8].nLevel,
    tSwitchOverTime := GVL_StreetLamps.tSwitchOverTime,
    bMemoryModeOn := GVL_StreetLamps.bMemoryModeOn,
    nOnValueWithoutMemoryMode := GVL_StreetLamps.nOnValueWithoutMemoryMode,
    nAddr := GVL_IO.arrStreetLamps[8].nAddrShort2,
    eAddrType := eDALIV2AddrTypeShort,
    nMasterDevAddr := GVL_StreetLamps.nMasterDevAddr,
    tCycleActualLevelMasterDev := GVL_StreetLamps.tCycleActualLevelMasterDev,
    stCommandBuffer := GVL_IO.stCommandBuffer_RB3); // FB_DALIV2Dimmer2Switch
fbDALIV2Dimmer2Switch_RB3_1(
    bSetDimmValue := GVL_StreetLamps.bSetDimmValue,
    nDimmValue := GVL_IO.arrStreetLamps[8].nLevel,
    tSwitchOverTime := GVL_StreetLamps.tSwitchOverTime,
    bMemoryModeOn := GVL_StreetLamps.bMemoryModeOn,
    nOnValueWithoutMemoryMode := GVL_StreetLamps.nOnValueWithoutMemoryMode,
    nAddr := GVL_IO.arrStreetLamps[8].nAddrShort1,
    eAddrType := eDALIV2AddrTypeShort,
    nMasterDevAddr := GVL_StreetLamps.nMasterDevAddr,
    tCycleActualLevelMasterDev := GVL_StreetLamps.tCycleActualLevelMasterDev,
    stCommandBuffer := GVL_IO.stCommandBuffer_RB3); // FB_DALIV2Dimmer2Switch
nActualLEvelMasterDev_2 := fbDALIV2Dimmer2Switch_RB3_2.nActualLevelMasterDev;
fbDALIV2Dimmer2Switch_RB3_3(
    bSetDimmValue := GVL_StreetLamps.bSetDimmValue,
    nDimmValue := GVL_IO.arrStreetLamps[9].nLevel,
    tSwitchOverTime := GVL_StreetLamps.tSwitchOverTime,
    bMemoryModeOn := GVL_StreetLamps.bMemoryModeOn,
    nOnValueWithoutMemoryMode := GVL_StreetLamps.nOnValueWithoutMemoryMode,
    nAddr := GVL_IO.arrStreetLamps[9].nAddrShort1,
    eAddrType := eDALIV2AddrTypeShort,
    nMasterDevAddr := GVL_StreetLamps.nMasterDevAddr,
    tCycleActualLevelMasterDev := GVL_StreetLamps.tCycleActualLevelMasterDev,
    stCommandBuffer := GVL_IO.stCommandBuffer_RB3); // FB_DALIV2Dimmer2Switch
bBusy_2 := fbDALIV2Dimmer2Switch_RB3_2.bBusy;
nActualLEvelMasterDev_1 := fbDALIV2Dimmer2Switch_RB3_1.nActualLevelMasterDev;
bBusy_1 := fbDALIV2Dimmer2Switch_RB3_1.bBusy;
bError_2 := fbDALIV2Dimmer2Switch_RB3_2.bError;
bError_1 := fbDALIV2Dimmer2Switch_RB3_1.bError;
nErrorId_2 := fbDALIV2Dimmer2Switch_RB3_2.nErrorId;
nActualLEvelMasterDev_3 := fbDALIV2Dimmer2Switch_RB3_3.nActualLevelMasterDev;
bBusy_3 := fbDALIV2Dimmer2Switch_RB3_3.bBusy;
nErrorId_1 := fbDALIV2Dimmer2Switch_RB3_1.nErrorId;
bError_3 := fbDALIV2Dimmer2Switch_RB3_3.bError;
nErrorId_3 := fbDALIV2Dimmer2Switch_RB3_3.nErrorId;
fbDALIV2Dimmer2Switch_RB3_4(
    bSetDimmValue := GVL_StreetLamps.bSetDimmValue,
    nDimmValue := GVL_IO.arrStreetLamps[9].nLevel,
    tSwitchOverTime := GVL_StreetLamps.tSwitchOverTime,
    bMemoryModeOn := GVL_StreetLamps.bMemoryModeOn,
    nOnValueWithoutMemoryMode := GVL_StreetLamps.nOnValueWithoutMemoryMode,
    nAddr := GVL_IO.arrStreetLamps[9].nAddrShort2,
    eAddrType := eDALIV2AddrTypeShort,
    nMasterDevAddr := GVL_StreetLamps.nMasterDevAddr,
    tCycleActualLevelMasterDev := GVL_StreetLamps.tCycleActualLevelMasterDev,
    stCommandBuffer := GVL_IO.stCommandBuffer_RB3); // FB_DALIV2Dimmer2Switch
nActualLEvelMasterDev_4 := fbDALIV2Dimmer2Switch_RB3_4.nActualLevelMasterDev;
bBusy_4 := fbDALIV2Dimmer2Switch_RB3_4.bBusy;
bError_4 := fbDALIV2Dimmer2Switch_RB3_4.bError;
nErrorId_4 := fbDALIV2Dimmer2Switch_RB3_4.nErrorId;
fbDALIV2Dimmer2Switch_RB3_5(
    bSetDimmValue := GVL_StreetLamps.bSetDimmValue,
    nDimmValue := GVL_IO.arrStreetLamps[10].nLevel,
    tSwitchOverTime := GVL_StreetLamps.tSwitchOverTime,
    bMemoryModeOn := GVL_StreetLamps.bMemoryModeOn,
    nOnValueWithoutMemoryMode := GVL_StreetLamps.nOnValueWithoutMemoryMode,
    nAddr := GVL_IO.arrStreetLamps[10].nAddrShort1,
    eAddrType := eDALIV2AddrTypeShort,
    nMasterDevAddr := GVL_StreetLamps.nMasterDevAddr,
    tCycleActualLevelMasterDev := GVL_StreetLamps.tCycleActualLevelMasterDev,
    stCommandBuffer := GVL_IO.stCommandBuffer_RB3); // FB_DALIV2Dimmer2Switch
nActualLEvelMasterDev_5 := fbDALIV2Dimmer2Switch_RB3_5.nActualLevelMasterDev;
bBusy_5 := fbDALIV2Dimmer2Switch_RB3_5.bBusy;
bError_5 := fbDALIV2Dimmer2Switch_RB3_5.bError;
nErrorId_5 := fbDALIV2Dimmer2Switch_RB3_5.nErrorId;
fbDALIV2Dimmer2Switch_RB3_6(
    bSetDimmValue := GVL_StreetLamps.bSetDimmValue,
    nDimmValue := GVL_IO.arrStreetLamps[10].nLevel,
    tSwitchOverTime := GVL_StreetLamps.tSwitchOverTime,
    bMemoryModeOn := GVL_StreetLamps.bMemoryModeOn,
    nOnValueWithoutMemoryMode := GVL_StreetLamps.nOnValueWithoutMemoryMode,
    nAddr := GVL_IO.arrStreetLamps[10].nAddrShort2,
    eAddrType := eDALIV2AddrTypeShort,
    nMasterDevAddr := GVL_StreetLamps.nMasterDevAddr,
    tCycleActualLevelMasterDev := GVL_StreetLamps.tCycleActualLevelMasterDev,
    stCommandBuffer := GVL_IO.stCommandBuffer_RB3); // FB_DALIV2Dimmer2Switch
nActualLEvelMasterDev_6 := fbDALIV2Dimmer2Switch_RB3_6.nActualLevelMasterDev;
bBusy_6 := fbDALIV2Dimmer2Switch_RB3_6.bBusy;
bError_6 := fbDALIV2Dimmer2Switch_RB3_6.bError;
nErrorId_6 := fbDALIV2Dimmer2Switch_RB3_6.nErrorId;

END_PROGRAM

// ---- POUs/DimmersStreetLamps/P_Dimmers_Broadcast.TcPOU
PROGRAM P_Dimmers_Broadcast
VAR
	fbDALIV2Dimmer2Switch_RB1		: FB_DALIV2Dimmer2Switch;
	nActualLEvelMasterDev_1			: BYTE;
	bBusy_1							: BOOL;
	bError_1						: BOOL;
	nErrorId_1						: UDINT;
	
	
	fbDALIV2Dimmer2Switch_RB2		: FB_DALIV2Dimmer2Switch;
	nActualLEvelMasterDev_2			: BYTE;
	bBusy_2							: BOOL;
	bError_2						: BOOL;
	nErrorId_2						: UDINT;
	
	
	fbDALIV2Dimmer2Switch_RB3		: FB_DALIV2Dimmer2Switch;
	nActualLEvelMasterDev_3			: BYTE;
	bBusy_3							: BOOL;
	bError_3						: BOOL;
	nErrorId_3						: UDINT;
END_VAR

fbDALIV2Dimmer2Switch_RB2(
    bSetDimmValue := GVL_StreetLamps.bSetDimmValue_B,
    nDimmValue := GVL_StreetLamps.nDimmValue_B,
    tSwitchOverTime := GVL_StreetLamps.tSwitchOverTime_B,
    bMemoryModeOn := GVL_StreetLamps.bMemoryModeOn_B,
    nOnValueWithoutMemoryMode := GVL_StreetLamps.nOnValueWithoutMemoryMode_B,
    nAddr := 0,
    eAddrType := eDALIV2AddrTypeBroadcast,
    nMasterDevAddr := GVL_StreetLamps.nMasterDevAddr_B,
    tCycleActualLevelMasterDev := GVL_StreetLamps.tCycleActualLevelMasterDev_B,
    stCommandBuffer := GVL_IO.stCommandBuffer_RB2); // FB_DALIV2Dimmer2Switch
fbDALIV2Dimmer2Switch_RB1(
    bSetDimmValue := GVL_StreetLamps.bSetDimmValue_B,
    nDimmValue := GVL_StreetLamps.nDimmValue_B,
    tSwitchOverTime := GVL_StreetLamps.tSwitchOverTime_B,
    bMemoryModeOn := GVL_StreetLamps.bMemoryModeOn_B,
    nOnValueWithoutMemoryMode := GVL_StreetLamps.nOnValueWithoutMemoryMode_B,
    nAddr := 0,
    eAddrType := eDALIV2AddrTypeBroadcast,
    nMasterDevAddr := GVL_StreetLamps.nMasterDevAddr_B,
    tCycleActualLevelMasterDev := GVL_StreetLamps.tCycleActualLevelMasterDev_B,
    stCommandBuffer := GVL_IO.stCommandBuffer_RB1); // FB_DALIV2Dimmer2Switch
nActualLEvelMasterDev_2 := fbDALIV2Dimmer2Switch_RB2.nActualLevelMasterDev;
bBusy_2 := fbDALIV2Dimmer2Switch_RB2.bBusy;
nActualLEvelMasterDev_1 := fbDALIV2Dimmer2Switch_RB1.nActualLevelMasterDev;
fbDALIV2Dimmer2Switch_RB3(
    bSetDimmValue := GVL_StreetLamps.bSetDimmValue_B,
    nDimmValue := GVL_StreetLamps.nDimmValue_B,
    tSwitchOverTime := GVL_StreetLamps.tSwitchOverTime_B,
    bMemoryModeOn := GVL_StreetLamps.bMemoryModeOn_B,
    nOnValueWithoutMemoryMode := GVL_StreetLamps.nOnValueWithoutMemoryMode_B,
    nAddr := 0,
    eAddrType := eDALIV2AddrTypeBroadcast,
    nMasterDevAddr := GVL_StreetLamps.nMasterDevAddr_B,
    tCycleActualLevelMasterDev := GVL_StreetLamps.tCycleActualLevelMasterDev_B,
    stCommandBuffer := GVL_IO.stCommandBuffer_RB3); // FB_DALIV2Dimmer2Switch
bBusy_1 := fbDALIV2Dimmer2Switch_RB1.bBusy;
bError_2 := fbDALIV2Dimmer2Switch_RB2.bError;
bError_1 := fbDALIV2Dimmer2Switch_RB1.bError;
nErrorId_2 := fbDALIV2Dimmer2Switch_RB2.nErrorId;
nErrorId_1 := fbDALIV2Dimmer2Switch_RB1.nErrorId;
bBusy_3 := fbDALIV2Dimmer2Switch_RB3.bBusy;
nActualLEvelMasterDev_3 := fbDALIV2Dimmer2Switch_RB3.nActualLevelMasterDev;
bError_3 := fbDALIV2Dimmer2Switch_RB3.bError;
nErrorId_3 := fbDALIV2Dimmer2Switch_RB3.nErrorId;

END_PROGRAM

// ---- POUs/BACnetControl/P_BACnet_ActualLevel.TcPOU
PROGRAM P_BACnet_ActualLevel
VAR
	i					: INT := 0;		//for loop counter
	arrActualLevel		: ARRAY [1..10] OF REAL;
	
	ton_Execute			: TON;
	
	fbDALIV2QueryActualLevel_1	 	: FB_DALIV2QueryActualLevel;
	fbDALIV2QueryActualLevel_2	 	: FB_DALIV2QueryActualLevel;
	fbDALIV2QueryActualLevel_3	 	: FB_DALIV2QueryActualLevel;
	fbDALIV2QueryActualLevel_4	 	: FB_DALIV2QueryActualLevel;
	fbDALIV2QueryActualLevel_5	 	: FB_DALIV2QueryActualLevel;
	fbDALIV2QueryActualLevel_6	 	: FB_DALIV2QueryActualLevel;
	fbDALIV2QueryActualLevel_7	 	: FB_DALIV2QueryActualLevel;
	fbDALIV2QueryActualLevel_8	 	: FB_DALIV2QueryActualLevel;
	fbDALIV2QueryActualLevel_9	 	: FB_DALIV2QueryActualLevel;
	fbDALIV2QueryActualLevel_10	 	: FB_DALIV2QueryActualLevel;
END_VAR

ton_Execute(IN := NOT ton_Execute.Q, PT := T#100MS);

fbDALIV2QueryActualLevel_1(
	bStart:= ton_Execute.Q, 
	nAddr:= GVL_IO.arrStreetLamps[1].nAddrShort1, 
	eAddrType:= eDALIV2AddrTypeShort, 
	eCommandPriority:= eDALIV2CommandPriorityLow,  
	stCommandBuffer:= GVL_IO.stCommandBuffer_RB1);

fbDALIV2QueryActualLevel_2(
	bStart:= ton_Execute.Q, 
	nAddr:= GVL_IO.arrStreetLamps[2].nAddrShort1, 
	eAddrType:= eDALIV2AddrTypeShort, 
	eCommandPriority:= eDALIV2CommandPriorityLow,  
	stCommandBuffer:= GVL_IO.stCommandBuffer_RB1);

fbDALIV2QueryActualLevel_3(
	bStart:= ton_Execute.Q, 
	nAddr:= GVL_IO.arrStreetLamps[3].nAddrShort1, 
	eAddrType:= eDALIV2AddrTypeShort, 
	eCommandPriority:= eDALIV2CommandPriorityLow,  
	stCommandBuffer:= GVL_IO.stCommandBuffer_RB1);

fbDALIV2QueryActualLevel_4(
	bStart:= ton_Execute.Q, 
	nAddr:= GVL_IO.arrStreetLamps[4].nAddrShort1, 
	eAddrType:= eDALIV2AddrTypeShort, 
	eCommandPriority:= eDALIV2CommandPriorityLow,  
	stCommandBuffer:= GVL_IO.stCommandBuffer_RB2);

fbDALIV2QueryActualLevel_5(
	bStart:= ton_Execute.Q, 
	nAddr:= GVL_IO.arrStreetLamps[5].nAddrShort1, 
	eAddrType:= eDALIV2AddrTypeShort, 
	eCommandPriority:= eDALIV2CommandPriorityLow,  
	stCommandBuffer:= GVL_IO.stCommandBuffer_RB2);

fbDALIV2QueryActualLevel_6(
	bStart:= ton_Execute.Q, 
	nAddr:= GVL_IO.arrStreetLamps[6].nAddrShort1, 
	eAddrType:= eDALIV2AddrTypeShort, 
	eCommandPriority:= eDALIV2CommandPriorityLow,  
	stCommandBuffer:= GVL_IO.stCommandBuffer_RB2);

fbDALIV2QueryActualLevel_7(
	bStart:= ton_Execute.Q, 
	nAddr:= GVL_IO.arrStreetLamps[7].nAddrShort1, 
	eAddrType:= eDALIV2AddrTypeShort, 
	eCommandPriority:= eDALIV2CommandPriorityLow,  
	stCommandBuffer:= GVL_IO.stCommandBuffer_RB2);

fbDALIV2QueryActualLevel_8(
	bStart:= ton_Execute.Q, 
	nAddr:= GVL_IO.arrStreetLamps[8].nAddrShort1, 
	eAddrType:= eDALIV2AddrTypeShort, 
	eCommandPriority:= eDALIV2CommandPriorityLow,  
	stCommandBuffer:= GVL_IO.stCommandBuffer_RB3);

fbDALIV2QueryActualLevel_9(
	bStart:= ton_Execute.Q, 
	nAddr:= GVL_IO.arrStreetLamps[9].nAddrShort1, 
	eAddrType:= eDALIV2AddrTypeShort, 
	eCommandPriority:= eDALIV2CommandPriorityLow,  
	stCommandBuffer:= GVL_IO.stCommandBuffer_RB3);

fbDALIV2QueryActualLevel_10(
	bStart:= ton_Execute.Q, 
	nAddr:= GVL_IO.arrStreetLamps[10].nAddrShort1, 
	eAddrType:= eDALIV2AddrTypeShort, 
	eCommandPriority:= eDALIV2CommandPriorityLow,  
	stCommandBuffer:= GVL_IO.stCommandBuffer_RB3);

	
//rewrite data to BACnet objects
fbBACnet_AV_SL_ActualLevel_1(Device := Device, bEnablePV := TRUE, bNullPV := FALSE, fPV := fbDALIV2QueryActualLevel_1.nActualLevel);
fbBACnet_AV_SL_ActualLevel_2(Device := Device, bEnablePV := TRUE, bNullPV := FALSE, fPV := fbDALIV2QueryActualLevel_2.nActualLevel);
fbBACnet_AV_SL_ActualLevel_3(Device := Device, bEnablePV := TRUE, bNullPV := FALSE, fPV := fbDALIV2QueryActualLevel_3.nActualLevel);
fbBACnet_AV_SL_ActualLevel_4(Device := Device, bEnablePV := TRUE, bNullPV := FALSE, fPV := fbDALIV2QueryActualLevel_4.nActualLevel);
fbBACnet_AV_SL_ActualLevel_5(Device := Device, bEnablePV := TRUE, bNullPV := FALSE, fPV := fbDALIV2QueryActualLevel_5.nActualLevel);
fbBACnet_AV_SL_ActualLevel_6(Device := Device, bEnablePV := TRUE, bNullPV := FALSE, fPV := fbDALIV2QueryActualLevel_6.nActualLevel);
fbBACnet_AV_SL_ActualLevel_7(Device := Device, bEnablePV := TRUE, bNullPV := FALSE, fPV := fbDALIV2QueryActualLevel_7.nActualLevel);
fbBACnet_AV_SL_ActualLevel_8(Device := Device, bEnablePV := TRUE, bNullPV := FALSE, fPV := fbDALIV2QueryActualLevel_8.nActualLevel);
fbBACnet_AV_SL_ActualLevel_9(Device := Device, bEnablePV := TRUE, bNullPV := FALSE, fPV := fbDALIV2QueryActualLevel_9.nActualLevel);
fbBACnet_AV_SL_ActualLevel_10(Device := Device, bEnablePV := TRUE, bNullPV := FALSE, fPV := fbDALIV2QueryActualLevel_10.nActualLevel);

END_PROGRAM

// ---- POUs/BACnetControl/P_BACnet_Error.TcPOU
PROGRAM P_BACnet_Error
VAR
	i					: INT := 0;		//for loop counter
	arrLampFailure		: ARRAY [1..10] OF BOOL;
	dwLampFailure		: DWORD;
	rLampFailure		: REAL;
	
	ton_Execute			: TON;
	
	fbDALIV2QueryLampFailure_1		: FB_DALIV2QueryLampFailure;
	fbDALIV2QueryLampFailure_2		: FB_DALIV2QueryLampFailure;
	fbDALIV2QueryLampFailure_3		: FB_DALIV2QueryLampFailure;
	fbDALIV2QueryLampFailure_4		: FB_DALIV2QueryLampFailure;
	fbDALIV2QueryLampFailure_5		: FB_DALIV2QueryLampFailure;
	fbDALIV2QueryLampFailure_6		: FB_DALIV2QueryLampFailure;
	fbDALIV2QueryLampFailure_7		: FB_DALIV2QueryLampFailure;
	fbDALIV2QueryLampFailure_8		: FB_DALIV2QueryLampFailure;
	fbDALIV2QueryLampFailure_9		: FB_DALIV2QueryLampFailure;
	fbDALIV2QueryLampFailure_10		: FB_DALIV2QueryLampFailure;
	
	fbDALIV2QueryLampFailure_1_2		: FB_DALIV2QueryLampFailure;
	fbDALIV2QueryLampFailure_2_2		: FB_DALIV2QueryLampFailure;
	fbDALIV2QueryLampFailure_3_2		: FB_DALIV2QueryLampFailure;
	fbDALIV2QueryLampFailure_4_2		: FB_DALIV2QueryLampFailure;
	fbDALIV2QueryLampFailure_5_2		: FB_DALIV2QueryLampFailure;
	fbDALIV2QueryLampFailure_6_2		: FB_DALIV2QueryLampFailure;
	fbDALIV2QueryLampFailure_7_2		: FB_DALIV2QueryLampFailure;
	fbDALIV2QueryLampFailure_8_2		: FB_DALIV2QueryLampFailure;
	fbDALIV2QueryLampFailure_9_2		: FB_DALIV2QueryLampFailure;
	fbDALIV2QueryLampFailure_10_2		: FB_DALIV2QueryLampFailure;
	
END_VAR

//init ton timer
ton_Execute(IN := NOT ton_Execute.Q, PT := T#100MS);

//query first half of the lamp
fbDALIV2QueryLampFailure_1(
		bStart:= ton_Execute.Q, 
		nAddr:= GVL_IO.arrStreetLamps[1].nAddrShort1, 
		eAddrType:= eDALIV2AddrTypeShort, 
		eCommandPriority:= eDALIV2CommandPriorityLow,  
		stCommandBuffer:= GVL_IO.stCommandBuffer_RB1);

//query second half of the lamp
fbDALIV2QueryLampFailure_1_2(
		bStart:= ton_Execute.Q, 
		nAddr:= GVL_IO.arrStreetLamps[1].nAddrShort2, 
		eAddrType:= eDALIV2AddrTypeShort, 
		eCommandPriority:= eDALIV2CommandPriorityLow,  
		stCommandBuffer:= GVL_IO.stCommandBuffer_RB1);
		
		//query first half of the lamp
fbDALIV2QueryLampFailure_2(
		bStart:= ton_Execute.Q, 
		nAddr:= GVL_IO.arrStreetLamps[2].nAddrShort1, 
		eAddrType:= eDALIV2AddrTypeShort, 
		eCommandPriority:= eDALIV2CommandPriorityLow,  
		stCommandBuffer:= GVL_IO.stCommandBuffer_RB1);

//query second half of the lamp
fbDALIV2QueryLampFailure_2_2(
		bStart:= ton_Execute.Q, 
		nAddr:= GVL_IO.arrStreetLamps[2].nAddrShort2, 
		eAddrType:= eDALIV2AddrTypeShort, 
		eCommandPriority:= eDALIV2CommandPriorityLow,  
		stCommandBuffer:= GVL_IO.stCommandBuffer_RB1);
		
		//query first half of the lamp
fbDALIV2QueryLampFailure_3(
		bStart:= ton_Execute.Q, 
		nAddr:= GVL_IO.arrStreetLamps[3].nAddrShort1, 
		eAddrType:= eDALIV2AddrTypeShort, 
		eCommandPriority:= eDALIV2CommandPriorityLow,  
		stCommandBuffer:= GVL_IO.stCommandBuffer_RB1);

//query second half of the lamp
fbDALIV2QueryLampFailure_3_2(
		bStart:= ton_Execute.Q, 
		nAddr:= GVL_IO.arrStreetLamps[3].nAddrShort2, 
		eAddrType:= eDALIV2AddrTypeShort, 
		eCommandPriority:= eDALIV2CommandPriorityLow,  
		stCommandBuffer:= GVL_IO.stCommandBuffer_RB1);
		
		//query first half of the lamp
fbDALIV2QueryLampFailure_4(
		bStart:= ton_Execute.Q, 
		nAddr:= GVL_IO.arrStreetLamps[4].nAddrShort1, 
		eAddrType:= eDALIV2AddrTypeShort, 
		eCommandPriority:= eDALIV2CommandPriorityLow,  
		stCommandBuffer:= GVL_IO.stCommandBuffer_RB2);

//query second half of the lamp
fbDALIV2QueryLampFailure_4_2(
		bStart:= ton_Execute.Q, 
		nAddr:= GVL_IO.arrStreetLamps[4].nAddrShort2, 
		eAddrType:= eDALIV2AddrTypeShort, 
		eCommandPriority:= eDALIV2CommandPriorityLow,  
		stCommandBuffer:= GVL_IO.stCommandBuffer_RB2);
		
		//query first half of the lamp
fbDALIV2QueryLampFailure_5(
		bStart:= ton_Execute.Q, 
		nAddr:= GVL_IO.arrStreetLamps[5].nAddrShort1, 
		eAddrType:= eDALIV2AddrTypeShort, 
		eCommandPriority:= eDALIV2CommandPriorityLow,  
		stCommandBuffer:= GVL_IO.stCommandBuffer_RB2);

//query second half of the lamp
fbDALIV2QueryLampFailure_5_2(
		bStart:= ton_Execute.Q, 
		nAddr:= GVL_IO.arrStreetLamps[5].nAddrShort2, 
		eAddrType:= eDALIV2AddrTypeShort, 
		eCommandPriority:= eDALIV2CommandPriorityLow,  
		stCommandBuffer:= GVL_IO.stCommandBuffer_RB2);
		
		//query first half of the lamp
fbDALIV2QueryLampFailure_6(
		bStart:= ton_Execute.Q, 
		nAddr:= GVL_IO.arrStreetLamps[6].nAddrShort1, 
		eAddrType:= eDALIV2AddrTypeShort, 
		eCommandPriority:= eDALIV2CommandPriorityLow,  
		stCommandBuffer:= GVL_IO.stCommandBuffer_RB2);

//query second half of the lamp
fbDALIV2QueryLampFailure_6_2(
		bStart:= ton_Execute.Q, 
		nAddr:= GVL_IO.arrStreetLamps[6].nAddrShort2, 
		eAddrType:= eDALIV2AddrTypeShort, 
		eCommandPriority:= eDALIV2CommandPriorityLow,  
		stCommandBuffer:= GVL_IO.stCommandBuffer_RB2);
		
		//query first half of the lamp
fbDALIV2QueryLampFailure_7(
		bStart:= ton_Execute.Q, 
		nAddr:= GVL_IO.arrStreetLamps[7].nAddrShort1, 
		eAddrType:= eDALIV2AddrTypeShort, 
		eCommandPriority:= eDALIV2CommandPriorityLow,  
		stCommandBuffer:= GVL_IO.stCommandBuffer_RB2);

//query second half of the lamp
fbDALIV2QueryLampFailure_7_2(
		bStart:= ton_Execute.Q, 
		nAddr:= GVL_IO.arrStreetLamps[7].nAddrShort2, 
		eAddrType:= eDALIV2AddrTypeShort, 
		eCommandPriority:= eDALIV2CommandPriorityLow,  
		stCommandBuffer:= GVL_IO.stCommandBuffer_RB2);
		
		//query first half of the lamp
fbDALIV2QueryLampFailure_8(
		bStart:= ton_Execute.Q, 
		nAddr:= GVL_IO.arrStreetLamps[8].nAddrShort1, 
		eAddrType:= eDALIV2AddrTypeShort, 
		eCommandPriority:= eDALIV2CommandPriorityLow,  
		stCommandBuffer:= GVL_IO.stCommandBuffer_RB3);

//query second half of the lamp
fbDALIV2QueryLampFailure_8_2(
		bStart:= ton_Execute.Q, 
		nAddr:= GVL_IO.arrStreetLamps[8].nAddrShort2, 
		eAddrType:= eDALIV2AddrTypeShort, 
		eCommandPriority:= eDALIV2CommandPriorityLow,  
		stCommandBuffer:= GVL_IO.stCommandBuffer_RB3);
		
		//query first half of the lamp
fbDALIV2QueryLampFailure_9(
		bStart:= ton_Execute.Q, 
		nAddr:= GVL_IO.arrStreetLamps[9].nAddrShort1, 
		eAddrType:= eDALIV2AddrTypeShort, 
		eCommandPriority:= eDALIV2CommandPriorityLow,  
		stCommandBuffer:= GVL_IO.stCommandBuffer_RB3);

//query second half of the lamp
fbDALIV2QueryLampFailure_9_2(
		bStart:= ton_Execute.Q, 
		nAddr:= GVL_IO.arrStreetLamps[9].nAddrShort2, 
		eAddrType:= eDALIV2AddrTypeShort, 
		eCommandPriority:= eDALIV2CommandPriorityLow,  
		stCommandBuffer:= GVL_IO.stCommandBuffer_RB3);
		
		//query first half of the lamp
fbDALIV2QueryLampFailure_10(
		bStart:= ton_Execute.Q, 
		nAddr:= GVL_IO.arrStreetLamps[10].nAddrShort1, 
		eAddrType:= eDALIV2AddrTypeShort, 
		eCommandPriority:= eDALIV2CommandPriorityLow,  
		stCommandBuffer:= GVL_IO.stCommandBuffer_RB3);

//query second half of the lamp
fbDALIV2QueryLampFailure_10_2(
		bStart:= ton_Execute.Q, 
		nAddr:= GVL_IO.arrStreetLamps[10].nAddrShort2, 
		eAddrType:= eDALIV2AddrTypeShort, 
		eCommandPriority:= eDALIV2CommandPriorityLow,  
		stCommandBuffer:= GVL_IO.stCommandBuffer_RB3);



	
//convert arrLampFailure into pseudo-array in the form of a DWORD variable
dwLampFailure.0 := fbDALIV2QueryLampFailure_1.bLampFailure  OR fbDALIV2QueryLampFailure_1_2.bLampFailure;
dwLampFailure.1 := fbDALIV2QueryLampFailure_2.bLampFailure  OR fbDALIV2QueryLampFailure_2_2.bLampFailure;
dwLampFailure.2 := fbDALIV2QueryLampFailure_3.bLampFailure  OR fbDALIV2QueryLampFailure_3_2.bLampFailure;
dwLampFailure.3 := fbDALIV2QueryLampFailure_4.bLampFailure  OR fbDALIV2QueryLampFailure_4_2.bLampFailure;
dwLampFailure.4 := fbDALIV2QueryLampFailure_5.bLampFailure  OR fbDALIV2QueryLampFailure_5_2.bLampFailure;
dwLampFailure.5 := fbDALIV2QueryLampFailure_6.bLampFailure  OR fbDALIV2QueryLampFailure_6_2.bLampFailure;
dwLampFailure.6 := fbDALIV2QueryLampFailure_7.bLampFailure  OR fbDALIV2QueryLampFailure_7_2.bLampFailure;
dwLampFailure.7 := fbDALIV2QueryLampFailure_8.bLampFailure  OR fbDALIV2QueryLampFailure_8_2.bLampFailure;
dwLampFailure.8 := fbDALIV2QueryLampFailure_9.bLampFailure  OR fbDALIV2QueryLampFailure_9_2.bLampFailure;
dwLampFailure.9 := fbDALIV2QueryLampFailure_10.bLampFailure OR fbDALIV2QueryLampFailure_10_2.bLampFailure;

//type conversion from REAL to DWORD
rLampFailure := DWORD_TO_REAL(dwLampFailure);

//write rLampFailure to BACnet obcject present value
//thereby keep BACnet object instance alive
fbBACnet_AV_SL_Error(Device := Device, bEnablePV := TRUE, bNullPV := FALSE, fPV := rLampFailure);

END_PROGRAM

// ---- POUs/BACnetControl/P_BACnet_Level.TcPOU
PROGRAM P_BACnet_Level
VAR
	ton_DelayForBACnet		: TON;
END_VAR

//assign fPV value to BACnet object if individual lamp is not in manual mode
fbBACnet_AV_SL_Level_1(Device := Device, bEnablePV := TRUE, bNullPV := FALSE);
fbBACnet_AV_SL_Level_2(Device := Device, bEnablePV := TRUE, bNullPV := FALSE);
fbBACnet_AV_SL_Level_3(Device := Device, bEnablePV := TRUE, bNullPV := FALSE);
fbBACnet_AV_SL_Level_4(Device := Device, bEnablePV := TRUE, bNullPV := FALSE);
fbBACnet_AV_SL_Level_5(Device := Device, bEnablePV := TRUE, bNullPV := FALSE);
fbBACnet_AV_SL_Level_6(Device := Device, bEnablePV := TRUE, bNullPV := FALSE);
fbBACnet_AV_SL_Level_7(Device := Device, bEnablePV := TRUE, bNullPV := FALSE);
fbBACnet_AV_SL_Level_8(Device := Device, bEnablePV := TRUE, bNullPV := FALSE);
fbBACnet_AV_SL_Level_9(Device := Device, bEnablePV := TRUE, bNullPV := FALSE);
fbBACnet_AV_SL_Level_10(Device := Device, bEnablePV := TRUE, bNullPV := FALSE);

//dalay for BACnet to catch up PLC
ton_DelayForBACnet(IN := NOT ton_DelayForBACnet.Q, PT := T#100MS);
IF ton_DelayForBACnet.Q THEN
	//if fPV does not match fPresentValue AND lamp is not in manual mode - increment fPV by 1, to force update
	IF fbBACnet_AV_SL_Level_1.fPresentValue  <> fbBACnet_AV_SL_Level_1.fPV  AND NOT GVL_IO.arrStreetLamps[1].bManualCtrl  THEN fbBACnet_AV_SL_Level_1.fPV  := fbBACnet_AV_SL_Level_1.fPV + 1;  END_IF
	IF fbBACnet_AV_SL_Level_2.fPresentValue  <> fbBACnet_AV_SL_Level_2.fPV  AND NOT GVL_IO.arrStreetLamps[2].bManualCtrl  THEN fbBACnet_AV_SL_Level_2.fPV  := fbBACnet_AV_SL_Level_2.fPV + 1;  END_IF
	IF fbBACnet_AV_SL_Level_3.fPresentValue  <> fbBACnet_AV_SL_Level_3.fPV  AND NOT GVL_IO.arrStreetLamps[3].bManualCtrl  THEN fbBACnet_AV_SL_Level_3.fPV  := fbBACnet_AV_SL_Level_3.fPV + 1;  END_IF
	IF fbBACnet_AV_SL_Level_4.fPresentValue  <> fbBACnet_AV_SL_Level_4.fPV  AND NOT GVL_IO.arrStreetLamps[4].bManualCtrl  THEN fbBACnet_AV_SL_Level_4.fPV  := fbBACnet_AV_SL_Level_4.fPV + 1;  END_IF
	IF fbBACnet_AV_SL_Level_5.fPresentValue  <> fbBACnet_AV_SL_Level_5.fPV  AND NOT GVL_IO.arrStreetLamps[5].bManualCtrl  THEN fbBACnet_AV_SL_Level_5.fPV  := fbBACnet_AV_SL_Level_5.fPV + 1;  END_IF
	IF fbBACnet_AV_SL_Level_6.fPresentValue  <> fbBACnet_AV_SL_Level_6.fPV  AND NOT GVL_IO.arrStreetLamps[6].bManualCtrl  THEN fbBACnet_AV_SL_Level_6.fPV  := fbBACnet_AV_SL_Level_6.fPV + 1;  END_IF
	IF fbBACnet_AV_SL_Level_7.fPresentValue  <> fbBACnet_AV_SL_Level_7.fPV  AND NOT GVL_IO.arrStreetLamps[7].bManualCtrl  THEN fbBACnet_AV_SL_Level_7.fPV  := fbBACnet_AV_SL_Level_7.fPV + 1;  END_IF
	IF fbBACnet_AV_SL_Level_8.fPresentValue  <> fbBACnet_AV_SL_Level_8.fPV  AND NOT GVL_IO.arrStreetLamps[8].bManualCtrl  THEN fbBACnet_AV_SL_Level_8.fPV  := fbBACnet_AV_SL_Level_8.fPV + 1;  END_IF
	IF fbBACnet_AV_SL_Level_9.fPresentValue  <> fbBACnet_AV_SL_Level_9.fPV  AND NOT GVL_IO.arrStreetLamps[9].bManualCtrl  THEN fbBACnet_AV_SL_Level_9.fPV  := fbBACnet_AV_SL_Level_9.fPV + 1;  END_IF
	IF fbBACnet_AV_SL_Level_10.fPresentValue <> fbBACnet_AV_SL_Level_10.fPV AND NOT GVL_IO.arrStreetLamps[10].bManualCtrl THEN fbBACnet_AV_SL_Level_10.fPV := fbBACnet_AV_SL_Level_10.fPV + 1; END_IF
END_IF

//rewrite present value to street lamp structures
 GVL_IO.arrStreetLamps[1].nLevel := REAL_TO_BYTE(fbBACnet_AV_SL_Level_1.fPresentValue);
 GVL_IO.arrStreetLamps[2].nLevel := REAL_TO_BYTE(fbBACnet_AV_SL_Level_2.fPresentValue);
 GVL_IO.arrStreetLamps[3].nLevel := REAL_TO_BYTE(fbBACnet_AV_SL_Level_3.fPresentValue);
 GVL_IO.arrStreetLamps[4].nLevel := REAL_TO_BYTE(fbBACnet_AV_SL_Level_4.fPresentValue);
 GVL_IO.arrStreetLamps[5].nLevel := REAL_TO_BYTE(fbBACnet_AV_SL_Level_5.fPresentValue);
 GVL_IO.arrStreetLamps[6].nLevel := REAL_TO_BYTE(fbBACnet_AV_SL_Level_6.fPresentValue);
 GVL_IO.arrStreetLamps[7].nLevel := REAL_TO_BYTE(fbBACnet_AV_SL_Level_7.fPresentValue);
 GVL_IO.arrStreetLamps[8].nLevel := REAL_TO_BYTE(fbBACnet_AV_SL_Level_8.fPresentValue);
 GVL_IO.arrStreetLamps[9].nLevel := REAL_TO_BYTE(fbBACnet_AV_SL_Level_9.fPresentValue);
 GVL_IO.arrStreetLamps[10].nLevel := REAL_TO_BYTE(fbBACnet_AV_SL_Level_10.fPresentValue);

END_PROGRAM

// ---- POUs/BACnetControl/P_BACnet_Manual.TcPOU
PROGRAM P_BACnet_Manual
VAR
	dwManual		: DWORD;
	
	rtReset			: R_TRIG;
	iSelector		: INT := 0;
	
	ton_DelayForBACnet	: TON;
END_VAR

//keep BACnet object instance alive
fbBACnet_AV_SL_Manual(Device := Device, bEnablePV := TRUE, bNullPV := FALSE);

//init rising edge initialization
rtReset(CLK := bBACnet_ResetManual);
//if rising edge occures
IF rtReset.Q THEN
	//set selector to 10
	iSelector := 10;
END_IF

CASE iSelector OF
	0:	//idle
		;	//do nothing
	10:
		fbBACnet_AV_SL_Manual.fPV := DWORD_TO_REAL(2#0001000000000000);
		iSelector := 20;
	20:
		//dalay for BACnet to catch up PLC
		ton_DelayForBACnet(IN := NOT ton_DelayForBACnet.Q, PT := T#100MS);
		IF ton_DelayForBACnet.Q THEN
			//if fPresentValue and fPV are different
			IF fbBACnet_AV_SL_Manual.fPresentValue <> fbBACnet_AV_SL_Manual.fPV THEN
				//increment fPV by 2#0001000000000000 to force the change of fPresentValue
				fbBACnet_AV_SL_Manual.fPV := fbBACnet_AV_SL_Manual.fPV + DWORD_TO_REAL(2#0001000000000000);
			ELSE
				bBACnet_ResetManual := FALSE;
				iSelector := 0;
			END_IF
		END_IF
END_CASE


//read REAL data from BACnet object
//and convert them to DWORD
dwManual := REAL_TO_DWORD(fbBACnet_AV_SL_Manual.fPresentValue);

//assign manual control flags
GVL_IO.arrStreetLamps[1].bManualCtrl := dwManual.0;
GVL_IO.arrStreetLamps[2].bManualCtrl := dwManual.1;
GVL_IO.arrStreetLamps[3].bManualCtrl := dwManual.2;
GVL_IO.arrStreetLamps[4].bManualCtrl := dwManual.3;
GVL_IO.arrStreetLamps[5].bManualCtrl := dwManual.4;
GVL_IO.arrStreetLamps[6].bManualCtrl := dwManual.5;
GVL_IO.arrStreetLamps[7].bManualCtrl := dwManual.6;
GVL_IO.arrStreetLamps[8].bManualCtrl := dwManual.7;
GVL_IO.arrStreetLamps[9].bManualCtrl := dwManual.8;
GVL_IO.arrStreetLamps[10].bManualCtrl := dwManual.9;

END_PROGRAM

// ---- POUs/BACnetControl/P_BACnet_Motion.TcPOU
PROGRAM P_BACnet_Motion
VAR
	dwMotion	: DWORD;	//pseudo-array for storing motion (BV) information
	rMotion		: REAL;		//dwMotion converted to REAL
END_VAR

//read motion sensor's flags and combine them into DWORD (pseudo-array)
dwMotion.0 := GVL_IO.arrStreetLamps[1].bMotionFlag;
dwMotion.1 := GVL_IO.arrStreetLamps[2].bMotionFlag;
dwMotion.2 := GVL_IO.arrStreetLamps[3].bMotionFlag;
dwMotion.3 := GVL_IO.arrStreetLamps[4].bMotionFlag;
dwMotion.4 := GVL_IO.arrStreetLamps[5].bMotionFlag;
dwMotion.5 := GVL_IO.arrStreetLamps[6].bMotionFlag;
dwMotion.6 := GVL_IO.arrStreetLamps[7].bMotionFlag;
dwMotion.7 := GVL_IO.arrStreetLamps[8].bMotionFlag;
dwMotion.8 := GVL_IO.arrStreetLamps[9].bMotionFlag;
dwMotion.9 := GVL_IO.arrStreetLamps[10].bMotionFlag;

//type conversion from DWORD to REAL
rMotion := DWORD_TO_REAL(dwMotion);

//write rMotion to BACnet obcject present value
//thereby keep BACnet object instance alive
fbBACnet_AV_SL_Motion(Device := Device, bEnablePV := TRUE, bNullPV := FALSE, fPV := rMotion);

END_PROGRAM

// ---- POUs/BACnetControl/P_BACnet_Scene.TcPOU
PROGRAM P_BACnet_Scene
VAR
END_VAR

//keep BACnet object alive
fbBACnet_AV_SL_Scene(Device := Device, bEnablePV := TRUE, bNullPV := FALSE);

END_PROGRAM

// ---- POUs/P_AutoMode_Old_Broadcast.TcPOU
PROGRAM P_AutoMode_Old_Broadcast
VAR
END_VAR

//if it is a night
IF F_IsNight() THEN
	//turn all lights full ON
	GVL_StreetLamps.nDimmValue_B := 255;
ELSE //it is a day
	//turn all lights OFF
	GVL_StreetLamps.nDimmValue_B := 0;
END_IF

END_PROGRAM
